LIN {X 0,Y 683.026,Z 572.337,A -85,B 0,C 180,E1 -4274.214,E2 -4274.214} C_VEL
LIN {X 0,Y 683.001,Z 572.333,A -85,B 0,C 180,E1 -4276.73,E2 -4276.73} C_VEL
LIN {X 0,Y 683.022,Z 572.332,A -85,B 0,C 180,E1 -4279.365,E2 -4279.365} C_VEL
LIN {X 0,Y 682.974,Z 572.347,A -85,B 0,C 180,E1 -4282.023,E2 -4282.023} C_VEL
LIN {X 0,Y 683,Z 572.34,A -85,B 0,C 180,E1 -4284.229,E2 -4284.229} C_VEL
LIN {X 0,Y 682.988,Z 572.339,A -85,B 0,C 180,E1 -4286.372,E2 -4286.372} C_VEL
LIN {X 0,Y 683.015,Z 572.334,A -85,B 0,C 180,E1 -4288.466,E2 -4288.466} C_VEL
LIN {X 0,Y 682.998,Z 572.334,A -85,B 0,C 180,E1 -4291.184,E2 -4291.184} C_VEL
LIN {X 0,Y 682.965,Z 572.347,A -85,B 0,C 180,E1 -4293.832,E2 -4293.832} C_VEL
LIN {X 0,Y 682.994,Z 572.345,A -85,B 0,C 180,E1 -4295.887,E2 -4295.887} C_VEL
LIN {X 0,Y 683.01,Z 572.336,A -85,B 0,C 180,E1 -4298.335,E2 -4298.335} C_VEL
LIN {X 0,Y 683.033,Z 572.329,A -85,B 0,C 180,E1 -4300.843,E2 -4300.843} C_VEL
LIN {X 0,Y 682.992,Z 572.336,A -85,B 0,C 180,E1 -4303.313,E2 -4303.313} C_VEL
LIN {X 0,Y 682.988,Z 572.343,A -85,B 0,C 180,E1 -4305.751,E2 -4305.751} C_VEL
LIN {X 0,Y 683.006,Z 572.34,A -85,B 0,C 180,E1 -4308.165,E2 -4308.165} C_VEL
LIN {X 0,Y 683.046,Z 572.329,A -85,B 0,C 180,E1 -4310.557,E2 -4310.557} C_VEL
LIN {X 0,Y 683.043,Z 572.328,A -85,B 0,C 180,E1 -4312.932,E2 -4312.932} C_VEL
LIN {X 0,Y 683.01,Z 572.332,A -85,B 0,C 180,E1 -4314.704,E2 -4314.704} C_VEL
LIN {X 0,Y 682.952,Z 572.342,A -85,B 0,C 180,E1 -4316.472,E2 -4316.472} C_VEL
LIN {X 0,Y 683.121,Z 572.318,A -85,B 0,C 180,E1 -4318.825,E2 -4318.825} C_VEL
LIN {X 0,Y 683.102,Z 572.329,A -85,B 0,C 180,E1 -4321.763,E2 -4321.763} C_VEL
LIN {X 0,Y 683.07,Z 572.325,A -85,B 0,C 180,E1 -4324.706,E2 -4324.706} C_VEL
LIN {X 0,Y 683.037,Z 572.328,A -85,B 0,C 180,E1 -4327.069,E2 -4327.069} C_VEL
LIN {X 0,Y 683.062,Z 572.336,A -85,B 0,C 180,E1 -4330.04,E2 -4330.04} C_VEL
LIN {X 0,Y 683.032,Z 572.329,A -85,B 0,C 180,E1 -4333.039,E2 -4333.039} C_VEL
LIN {X 0,Y 683.005,Z 572.336,A -85,B 0,C 180,E1 -4335.464,E2 -4335.464} C_VEL
LIN {X 0,Y 682.987,Z 572.347,A -85,B 0,C 180,E1 -4337.919,E2 -4337.919} C_VEL
LIN {X 0,Y 682.965,Z 572.346,A -85,B 0,C 180,E1 -4339.782,E2 -4339.782} C_VEL
LIN {X 0,Y 682.975,Z 572.337,A -85,B 0,C 180,E1 -4342.628,E2 -4342.628} C_VEL
LIN {X 0,Y 682.991,Z 572.334,A -85,B 0,C 180,E1 -4344.865,E2 -4344.865} C_VEL
LIN {X 0,Y 682.98,Z 572.339,A -85,B 0,C 180,E1 -4347.484,E2 -4347.484} C_VEL
LIN {X 0,Y 682.979,Z 572.34,A -85,B 0,C 180,E1 -4349.49,E2 -4349.49} C_VEL
LIN {X 0,Y 682.971,Z 572.343,A -85,B 0,C 180,E1 -4352.229,E2 -4352.229} C_VEL
LIN {X 0,Y 682.965,Z 572.342,A -85,B 0,C 180,E1 -4354.338,E2 -4354.338} C_VEL
LIN {X 0,Y 682.944,Z 572.34,A -85,B 0,C 180,E1 -4356.871,E2 -4356.871} C_VEL
LIN {X 0,Y 682.965,Z 572.338,A -85,B 0,C 180,E1 -4358.79,E2 -4358.79} C_VEL
LIN {X 0,Y 682.959,Z 572.343,A -85,B 0,C 180,E1 -4361.523,E2 -4361.523} C_VEL
LIN {X 0,Y 682.988,Z 572.341,A -85,B 0,C 180,E1 -4364.217,E2 -4364.217} C_VEL
LIN {X 0,Y 682.936,Z 572.341,A -85,B 0,C 180,E1 -4366.736,E2 -4366.736} C_VEL
LIN {X 0,Y 682.97,Z 572.339,A -85,B 0,C 180,E1 -4369.37,E2 -4369.37} C_VEL
LIN {X 0,Y 682.965,Z 572.345,A -85,B 0,C 180,E1 -4372.158,E2 -4372.158} C_VEL
LIN {X 0,Y 682.961,Z 572.338,A -85,B 0,C 180,E1 -4374.947,E2 -4374.947} C_VEL
LIN {X 0,Y 682.985,Z 572.336,A -85,B 0,C 180,E1 -4377.242,E2 -4377.242} C_VEL
LIN {X 0,Y 682.949,Z 572.349,A -85,B 0,C 180,E1 -4379.831,E2 -4379.831} C_VEL
LIN {X 0,Y 682.954,Z 572.341,A -85,B 0,C 180,E1 -4382.515,E2 -4382.515} C_VEL
LIN {X 0,Y 682.986,Z 572.337,A -85,B 0,C 180,E1 -4385.135,E2 -4385.135} C_VEL
LIN {X 0,Y 682.994,Z 572.346,A -85,B 0,C 180,E1 -4388.215,E2 -4388.215} C_VEL
LIN {X 0,Y 683.856,Z 577.659,A -85,B 0,C 180,E1 -4388.993,E2 -4388.993} C_VEL
LIN {X 0,Y 683.698,Z 593.941,A -85,B 0,C 180,E1 -4391.173,E2 -4391.173} C_VEL
LIN {X 0,Y 683.385,Z 612.574,A -85,B 0,C 180,E1 -4393.629,E2 -4393.629} C_VEL
LIN {X 0,Y 683.159,Z 631.189,A -85,B 0,C 180,E1 -4396.058,E2 -4396.058} C_VEL
LIN {X 0,Y 682.934,Z 649.485,A -85,B 0,C 180,E1 -4398.426,E2 -4398.426} C_VEL
LIN {X 0,Y 683.89,Z 658.24,A -85,B 0,C 180,E1 -4398.536,E2 -4398.536} C_VEL
LIN {X 0,Y 683.613,Z 755.729,A -85,B 0,C 180,E1 -4399.57,E2 -4399.57} C_VEL
LIN {X 0,Y 683.524,Z 765.358,A -85,B 0,C 180,E1 -4399.735,E2 -4399.735} C_VEL
LIN {X 0,Y 683.504,Z 776.178,A -85,B 0,C 180,E1 -4400.004,E2 -4400.004} C_VEL
LIN {X 0,Y 683.404,Z 786.265,A -85,B 0,C 180,E1 -4400.338,E2 -4400.338} C_VEL
LIN {X 0,Y 683.279,Z 796.757,A -85,B 0,C 180,E1 -4400.783,E2 -4400.783} C_VEL
LIN {X 0,Y 683.151,Z 806.601,A -85,B 0,C 180,E1 -4401.302,E2 -4401.302} C_VEL
LIN {X 0,Y 682.995,Z 814.812,A -85,B 0,C 180,E1 -4401.819,E2 -4401.819} C_VEL
LIN {X 0,Y 682.831,Z 823.576,A -85,B 0,C 180,E1 -4402.485,E2 -4402.485} C_VEL
LIN {X 0,Y 682.732,Z 831.633,A -85,B 0,C 180,E1 -4403.224,E2 -4403.224} C_VEL
LIN {X 0,Y 682.647,Z 838.345,A -85,B 0,C 180,E1 -4403.963,E2 -4403.963} C_VEL
LIN {X 0,Y 682.561,Z 843.958,A -85,B 0,C 180,E1 -4404.701,E2 -4404.701} C_VEL
LIN {X 0,Y 682.519,Z 849.404,A -85,B 0,C 180,E1 -4405.586,E2 -4405.586} C_VEL
LIN {X 0,Y 682.471,Z 853.686,A -85,B 0,C 180,E1 -4406.47,E2 -4406.47} C_VEL
LIN {X 0,Y 682.508,Z 855.979,A -85,B 0,C 180,E1 -4407.059,E2 -4407.059} C_VEL
LIN {X 0,Y 682.422,Z 859.189,A -85,B 0,C 180,E1 -4408.236,E2 -4408.236} C_VEL
LIN {X 0,Y 682.405,Z 860.148,A -85,B 0,C 180,E1 -4408.824,E2 -4408.824} C_VEL
LIN {X 0,Y 682.375,Z 861,A -85,B 0,C 180,E1 -4410,E2 -4410} C_VEL
LIN {X 0,Y 682.406,Z 860.149,A -85,B 0,C 180,E1 -4411.176,E2 -4411.176} C_VEL
LIN {X 0,Y 682.423,Z 859.191,A -85,B 0,C 180,E1 -4411.765,E2 -4411.765} C_VEL
LIN {X 0,Y 682.508,Z 855.981,A -85,B 0,C 180,E1 -4412.941,E2 -4412.941} C_VEL
LIN {X 0,Y 682.475,Z 852.425,A -85,B 0,C 180,E1 -4413.825,E2 -4413.825} C_VEL
LIN {X 0,Y 682.558,Z 847.764,A -85,B 0,C 180,E1 -4414.709,E2 -4414.709} C_VEL
LIN {X 0,Y 682.601,Z 841.063,A -85,B 0,C 180,E1 -4415.694,E2 -4415.694} C_VEL
LIN {X 0,Y 682.667,Z 834.458,A -85,B 0,C 180,E1 -4416.481,E2 -4416.481} C_VEL
LIN {X 0,Y 682.799,Z 826.966,A -85,B 0,C 180,E1 -4417.219,E2 -4417.219} C_VEL
LIN {X 0,Y 682.918,Z 818.879,A -85,B 0,C 180,E1 -4417.885,E2 -4417.885} C_VEL
LIN {X 0,Y 683.048,Z 810.276,A -85,B 0,C 180,E1 -4418.477,E2 -4418.477} C_VEL
LIN {X 0,Y 683.207,Z 801.24,A -85,B 0,C 180,E1 -4418.995,E2 -4418.995} C_VEL
LIN {X 0,Y 683.361,Z 791.852,A -85,B 0,C 180,E1 -4419.439,E2 -4419.439} C_VEL
LIN {X 0,Y 683.439,Z 780.985,A -85,B 0,C 180,E1 -4419.848,E2 -4419.848} C_VEL
LIN {X 0,Y 683.513,Z 770.389,A -85,B 0,C 180,E1 -4420.152,E2 -4420.152} C_VEL
LIN {X 0,Y 683.657,Z 759.149,A -85,B 0,C 180,E1 -4420.38,E2 -4420.38} C_VEL
LIN {X 0,Y 683.695,Z 742.553,A -85,B 0,C 180,E1 -4420.584,E2 -4420.584} C_VEL
LIN {X 0,Y 683.821,Z 656.435,A -85,B 0,C 180,E1 -4421.484,E2 -4421.484} C_VEL
LIN {X 0,Y 682.934,Z 649.483,A -85,B 0,C 180,E1 -4421.575,E2 -4421.575} C_VEL
LIN {X 0,Y 683.16,Z 631.148,A -85,B 0,C 180,E1 -4423.943,E2 -4423.943} C_VEL
LIN {X 0,Y 683.411,Z 611.307,A -85,B 0,C 180,E1 -4426.524,E2 -4426.524} C_VEL
LIN {X 0,Y 683.768,Z 589.908,A -85,B 0,C 180,E1 -4429.339,E2 -4429.339} C_VEL
LIN {X 0,Y 683.834,Z 577.443,A -85,B 0,C 180,E1 -4431.008,E2 -4431.008} C_VEL
LIN {X 0,Y 682.983,Z 572.347,A -85,B 0,C 180,E1 -4431.746,E2 -4431.746} C_VEL
LIN {X 0,Y 682.954,Z 572.348,A -85,B 0,C 180,E1 -4434.22,E2 -4434.22} C_VEL
LIN {X 0,Y 682.968,Z 572.341,A -85,B 0,C 180,E1 -4436.841,E2 -4436.841} C_VEL
LIN {X 0,Y 682.969,Z 572.347,A -85,B 0,C 180,E1 -4439.491,E2 -4439.491} C_VEL
LIN {X 0,Y 682.972,Z 572.341,A -85,B 0,C 180,E1 -4442.229,E2 -4442.229} C_VEL
LIN {X 0,Y 682.979,Z 572.338,A -85,B 0,C 180,E1 -4444.87,E2 -4444.87} C_VEL
LIN {X 0,Y 682.963,Z 572.344,A -85,B 0,C 180,E1 -4447.236,E2 -4447.236} C_VEL
LIN {X 0,Y 682.955,Z 572.345,A -85,B 0,C 180,E1 -4449.717,E2 -4449.717} C_VEL
LIN {X 0,Y 682.985,Z 572.339,A -85,B 0,C 180,E1 -4451.807,E2 -4451.807} C_VEL
LIN {X 0,Y 682.996,Z 572.335,A -85,B 0,C 180,E1 -4454.217,E2 -4454.217} C_VEL
LIN {X 0,Y 683.006,Z 572.337,A -85,B 0,C 180,E1 -4456.73,E2 -4456.73} C_VEL
LIN {X 0,Y 683.028,Z 572.339,A -85,B 0,C 180,E1 -4459.365,E2 -4459.365} C_VEL
LIN {X 0,Y 682.977,Z 572.338,A -85,B 0,C 180,E1 -4462.157,E2 -4462.157} C_VEL
LIN {X 0,Y 683.018,Z 572.342,A -85,B 0,C 180,E1 -4464.95,E2 -4464.95} C_VEL
LIN {X 0,Y 683.017,Z 572.332,A -85,B 0,C 180,E1 -4467.773,E2 -4467.773} C_VEL
LIN {X 0,Y 682.996,Z 572.334,A -85,B 0,C 180,E1 -4469.833,E2 -4469.833} C_VEL
LIN {X 0,Y 683.027,Z 572.331,A -85,B 0,C 180,E1 -4471.876,E2 -4471.876} C_VEL
LIN {X 0,Y 682.998,Z 572.343,A -85,B 0,C 180,E1 -4474.486,E2 -4474.486} C_VEL
LIN {X 0,Y 683,Z 572.339,A -85,B 0,C 180,E1 -4477.064,E2 -4477.064} C_VEL
LIN {X 0,Y 682.981,Z 572.339,A -85,B 0,C 180,E1 -4479.592,E2 -4479.592} C_VEL
LIN {X 0,Y 683.01,Z 572.335,A -85,B 0,C 180,E1 -4481.463,E2 -4481.463} C_VEL
LIN {X 0,Y 682.992,Z 572.34,A -85,B 0,C 180,E1 -4483.925,E2 -4483.925} C_VEL
LIN {X 0,Y 683.015,Z 572.344,A -85,B 0,C 180,E1 -4486.357,E2 -4486.357} C_VEL
LIN {X 0,Y 683.015,Z 572.338,A -85,B 0,C 180,E1 -4488.764,E2 -4488.764} C_VEL
LIN {X 0,Y 683.058,Z 572.423,A -85,B 0,C 180,E1 -4490.929,E2 -4490.929} C_VEL
LIN {X 0,Y 683.487,Z 579.381,A -85,B 0,C 180,E1 -4492.048,E2 -4492.048} C_VEL
LIN {X 0,Y 683.242,Z 596.262,A -85,B 0,C 180,E1 -4494.706,E2 -4494.706} C_VEL
LIN {X 0,Y 682.99,Z 609.521,A -85,B 0,C 180,E1 -4496.766,E2 -4496.766} C_VEL
LIN {X 0,Y 682.853,Z 620.602,A -85,B 0,C 180,E1 -4498.475,E2 -4498.475} C_VEL
LIN {X 0,Y 683.914,Z 628.858,A -85,B 0,C 180,E1 -4498.588,E2 -4498.588} C_VEL
LIN {X 0,Y 683.517,Z 727.56,A -85,B 0,C 180,E1 -4499.633,E2 -4499.633} C_VEL
LIN {X 0,Y 683.418,Z 740.394,A -85,B 0,C 180,E1 -4499.89,E2 -4499.89} C_VEL
LIN {X 0,Y 683.336,Z 752.881,A -85,B 0,C 180,E1 -4500.257,E2 -4500.257} C_VEL
LIN {X 0,Y 683.323,Z 764.89,A -85,B 0,C 180,E1 -4500.734,E2 -4500.734} C_VEL
LIN {X 0,Y 683.123,Z 776.26,A -85,B 0,C 180,E1 -4501.322,E2 -4501.322} C_VEL
LIN {X 0,Y 682.987,Z 786.525,A -85,B 0,C 180,E1 -4501.983,E2 -4501.983} C_VEL
LIN {X 0,Y 682.762,Z 795.042,A -85,B 0,C 180,E1 -4502.646,E2 -4502.646} C_VEL
LIN {X 0,Y 682.683,Z 802.781,A -85,B 0,C 180,E1 -4503.382,E2 -4503.382} C_VEL
LIN {X 0,Y 682.531,Z 810.48,A -85,B 0,C 180,E1 -4504.267,E2 -4504.267} C_VEL
LIN {X 0,Y 682.532,Z 815.691,A -85,B 0,C 180,E1 -4505.004,E2 -4505.004} C_VEL
LIN {X 0,Y 682.498,Z 820.823,A -85,B 0,C 180,E1 -4505.89,E2 -4505.89} C_VEL
LIN {X 0,Y 682.465,Z 824.783,A -85,B 0,C 180,E1 -4506.778,E2 -4506.778} C_VEL
LIN {X 0,Y 682.403,Z 827.744,A -85,B 0,C 180,E1 -4507.668,E2 -4507.668} C_VEL
LIN {X 0,Y 682.391,Z 829.173,A -85,B 0,C 180,E1 -4508.262,E2 -4508.262} C_VEL
LIN {X 0,Y 682.414,Z 830.191,A -85,B 0,C 180,E1 -4508.856,E2 -4508.856} C_VEL
LIN {X 0,Y 682.438,Z 831,A -85,B 0,C 180,E1 -4510.048,E2 -4510.048} C_VEL
LIN {X 0,Y 682.389,Z 830.173,A -85,B 0,C 180,E1 -4511.246,E2 -4511.246} C_VEL
LIN {X 0,Y 682.396,Z 829.138,A -85,B 0,C 180,E1 -4511.846,E2 -4511.846} C_VEL
LIN {X 0,Y 682.448,Z 826.515,A -85,B 0,C 180,E1 -4512.824,E2 -4512.824} C_VEL
LIN {X 0,Y 682.443,Z 823.402,A -85,B 0,C 180,E1 -4513.654,E2 -4513.654} C_VEL
LIN {X 0,Y 682.509,Z 818.861,A -85,B 0,C 180,E1 -4514.562,E2 -4514.562} C_VEL
LIN {X 0,Y 682.562,Z 813.1,A -85,B 0,C 180,E1 -4515.474,E2 -4515.474} C_VEL
LIN {X 0,Y 682.66,Z 805.78,A -85,B 0,C 180,E1 -4516.389,E2 -4516.389} C_VEL
LIN {X 0,Y 682.765,Z 798.238,A -85,B 0,C 180,E1 -4517.154,E2 -4517.154} C_VEL
LIN {X 0,Y 682.922,Z 789.106,A -85,B 0,C 180,E1 -4517.92,E2 -4517.92} C_VEL
LIN {X 0,Y 683.022,Z 778.927,A -85,B 0,C 180,E1 -4518.614,E2 -4518.614} C_VEL
LIN {X 0,Y 683.166,Z 769.09,A -85,B 0,C 180,E1 -4519.153,E2 -4519.153} C_VEL
LIN {X 0,Y 683.38,Z 757.902,A -85,B 0,C 180,E1 -4519.651,E2 -4519.651} C_VEL
LIN {X 0,Y 683.455,Z 746.324,A -85,B 0,C 180,E1 -4520.04,E2 -4520.04} C_VEL
LIN {X 0,Y 683.581,Z 733.577,A -85,B 0,C 180,E1 -4520.349,E2 -4520.349} C_VEL
LIN {X 0,Y 683.672,Z 720.861,A -85,B 0,C 180,E1 -4520.542,E2 -4520.542} C_VEL
LIN {X 0,Y 683.853,Z 627.908,A -85,B 0,C 180,E1 -4521.513,E2 -4521.513} C_VEL
LIN {X 0,Y 682.833,Z 620.616,A -85,B 0,C 180,E1 -4521.611,E2 -4521.611} C_VEL
LIN {X 0,Y 682.975,Z 608.393,A -85,B 0,C 180,E1 -4523.492,E2 -4523.492} C_VEL
LIN {X 0,Y 682.356,Z 605.665,A -85,B 0,C 180,E1 -4523.928,E2 -4523.928} C_VEL
LIN {X 0,Y 676.758,Z 597.294,A -85,B 0,C 180,E1 -4525.373,E2 -4525.373} C_VEL
LIN {X 0,Y 676.16,Z 594.582,A -85,B 0,C 180,E1 -4525.816,E2 -4525.816} C_VEL
LIN {X 0,Y 676.414,Z 577.967,A -85,B 0,C 180,E1 -4528.446,E2 -4528.446} C_VEL
LIN {X 0,Y 675.969,Z 573.219,A -85,B 0,C 180,E1 -4529.233,E2 -4529.233} C_VEL
LIN {X 0,Y 675.971,Z 573.212,A -85,B 0,C 180,E1 -4531.205,E2 -4531.205} C_VEL
LIN {X 0,Y 675.962,Z 573.221,A -85,B 0,C 180,E1 -4534.025,E2 -4534.025} C_VEL
LIN {X 0,Y 675.942,Z 573.219,A -85,B 0,C 180,E1 -4536.204,E2 -4536.204} C_VEL
LIN {X 0,Y 675.938,Z 573.213,A -85,B 0,C 180,E1 -4538.996,E2 -4538.996} C_VEL
LIN {X 0,Y 675.972,Z 573.216,A -85,B 0,C 180,E1 -4541.749,E2 -4541.749} C_VEL
LIN {X 0,Y 675.985,Z 573.211,A -85,B 0,C 180,E1 -4544.359,E2 -4544.359} C_VEL
LIN {X 0,Y 675.946,Z 573.212,A -85,B 0,C 180,E1 -4546.849,E2 -4546.849} C_VEL
LIN {X 0,Y 675.967,Z 573.21,A -85,B 0,C 180,E1 -4549.246,E2 -4549.246} C_VEL
LIN {X 0,Y 675.937,Z 573.225,A -85,B 0,C 180,E1 -4551.957,E2 -4551.957} C_VEL
LIN {X 0,Y 675.946,Z 573.214,A -85,B 0,C 180,E1 -4554.528,E2 -4554.528} C_VEL
LIN {X 0,Y 675.946,Z 573.212,A -85,B 0,C 180,E1 -4557.071,E2 -4557.071} C_VEL
LIN {X 0,Y 676.001,Z 573.209,A -85,B 0,C 180,E1 -4559.488,E2 -4559.488} C_VEL
LIN {X 0,Y 675.948,Z 573.219,A -85,B 0,C 180,E1 -4562.205,E2 -4562.205} C_VEL
LIN {X 0,Y 675.945,Z 573.212,A -85,B 0,C 180,E1 -4564.858,E2 -4564.858} C_VEL
LIN {X 0,Y 675.976,Z 573.211,A -85,B 0,C 180,E1 -4567.456,E2 -4567.456} C_VEL
LIN {X 0,Y 675.936,Z 573.224,A -85,B 0,C 180,E1 -4570.003,E2 -4570.003} C_VEL
LIN {X 0,Y 675.997,Z 573.208,A -85,B 0,C 180,E1 -4572.513,E2 -4572.513} C_VEL
LIN {X 0,Y 675.997,Z 573.205,A -85,B 0,C 180,E1 -4574.987,E2 -4574.987} C_VEL
LIN {X 0,Y 675.997,Z 573.208,A -85,B 0,C 180,E1 -4577.432,E2 -4577.432} C_VEL
LIN {X 0,Y 676.01,Z 573.207,A -85,B 0,C 180,E1 -4580.457,E2 -4580.457} C_VEL
LIN {X 0,Y 676.011,Z 573.204,A -85,B 0,C 180,E1 -4582.857,E2 -4582.857} C_VEL
LIN {X 0,Y 676.046,Z 573.2,A -85,B 0,C 180,E1 -4585.245,E2 -4585.245} C_VEL
LIN {X 0,Y 676.106,Z 573.192,A -85,B 0,C 180,E1 -4588.813,E2 -4588.813} C_VEL
LIN {X 0,Y 676.086,Z 573.203,A -85,B 0,C 180,E1 -4591.781,E2 -4591.781} C_VEL
LIN {X 0,Y 676.046,Z 573.2,A -85,B 0,C 180,E1 -4594.754,E2 -4594.754} C_VEL
LIN {X 0,Y 676.011,Z 573.204,A -85,B 0,C 180,E1 -4597.142,E2 -4597.142} C_VEL
LIN {X 0,Y 675.986,Z 573.215,A -85,B 0,C 180,E1 -4600.146,E2 -4600.146} C_VEL
LIN {X 0,Y 676.012,Z 573.204,A -85,B 0,C 180,E1 -4603.176,E2 -4603.176} C_VEL
LIN {X 0,Y 676.008,Z 573.21,A -85,B 0,C 180,E1 -4605.628,E2 -4605.628} C_VEL
LIN {X 0,Y 675.976,Z 573.217,A -85,B 0,C 180,E1 -4608.111,E2 -4608.111} C_VEL
LIN {X 0,Y 675.954,Z 573.212,A -85,B 0,C 180,E1 -4610.629,E2 -4610.629} C_VEL
LIN {X 0,Y 675.962,Z 573.21,A -85,B 0,C 180,E1 -4613.189,E2 -4613.189} C_VEL
LIN {X 0,Y 675.928,Z 573.223,A -85,B 0,C 180,E1 -4615.8,E2 -4615.8} C_VEL
LIN {X 0,Y 675.958,Z 573.216,A -85,B 0,C 180,E1 -4618.263,E2 -4618.263} C_VEL
LIN {X 0,Y 675.995,Z 573.206,A -85,B 0,C 180,E1 -4620.682,E2 -4620.682} C_VEL
LIN {X 0,Y 675.96,Z 573.212,A -85,B 0,C 180,E1 -4623.312,E2 -4623.312} C_VEL
LIN {X 0,Y 675.978,Z 573.217,A -85,B 0,C 180,E1 -4626.077,E2 -4626.077} C_VEL
LIN {X 0,Y 675.937,Z 573.213,A -85,B 0,C 180,E1 -4628.997,E2 -4628.997} C_VEL
LIN {X 0,Y 675.97,Z 573.217,A -85,B 0,C 180,E1 -4631.75,E2 -4631.75} C_VEL
LIN {X 0,Y 675.984,Z 573.211,A -85,B 0,C 180,E1 -4634.36,E2 -4634.36} C_VEL
LIN {X 0,Y 675.944,Z 573.212,A -85,B 0,C 180,E1 -4636.85,E2 -4636.85} C_VEL
LIN {X 0,Y 675.966,Z 573.21,A -85,B 0,C 180,E1 -4639.246,E2 -4639.246} C_VEL
LIN {X 0,Y 675.938,Z 573.225,A -85,B 0,C 180,E1 -4641.957,E2 -4641.957} C_VEL
LIN {X 0,Y 675.946,Z 573.214,A -85,B 0,C 180,E1 -4644.529,E2 -4644.529} C_VEL
LIN {X 0,Y 675.946,Z 573.212,A -85,B 0,C 180,E1 -4647.072,E2 -4647.072} C_VEL
LIN {X 0,Y 676.002,Z 573.209,A -85,B 0,C 180,E1 -4649.489,E2 -4649.489} C_VEL
LIN {X 0,Y 675.944,Z 573.219,A -85,B 0,C 180,E1 -4652.205,E2 -4652.205} C_VEL
LIN {X 0,Y 675.947,Z 573.212,A -85,B 0,C 180,E1 -4654.859,E2 -4654.859} C_VEL
LIN {X 0,Y 675.977,Z 573.211,A -85,B 0,C 180,E1 -4657.456,E2 -4657.456} C_VEL
LIN {X 0,Y 675.937,Z 573.224,A -85,B 0,C 180,E1 -4660.004,E2 -4660.004} C_VEL
LIN {X 0,Y 675.958,Z 573.213,A -85,B 0,C 180,E1 -4662.512,E2 -4662.512} C_VEL
LIN {X 0,Y 675.945,Z 573.212,A -85,B 0,C 180,E1 -4664.986,E2 -4664.986} C_VEL
LIN {X 0,Y 675.984,Z 573.21,A -85,B 0,C 180,E1 -4667.432,E2 -4667.432} C_VEL
LIN {X 0,Y 676.031,Z 573.212,A -85,B 0,C 180,E1 -4669.855,E2 -4669.855} C_VEL
LIN {X 0,Y 676.011,Z 573.204,A -85,B 0,C 180,E1 -4672.858,E2 -4672.858} C_VEL
LIN {X 0,Y 676.013,Z 573.205,A -85,B 0,C 180,E1 -4675.245,E2 -4675.245} C_VEL
LIN {X 0,Y 676.107,Z 573.198,A -85,B 0,C 180,E1 -4678.219,E2 -4678.219} C_VEL
LIN {X 0,Y 676.095,Z 573.194,A -85,B 0,C 180,E1 -4681.187,E2 -4681.187} C_VEL
LIN {X 0,Y 676.053,Z 573.206,A -85,B 0,C 180,E1 -4684.159,E2 -4684.159} C_VEL
LIN {X 0,Y 676.026,Z 573.204,A -85,B 0,C 180,E1 -4686.545,E2 -4686.545} C_VEL
LIN {X 0,Y 676.015,Z 573.208,A -85,B 0,C 180,E1 -4689.543,E2 -4689.543} C_VEL
LIN {X 0,Y 675.944,Z 573.224,A -85,B 0,C 180,E1 -4691.961,E2 -4691.961} C_VEL
LIN {X 0,Y 675.945,Z 573.216,A -85,B 0,C 180,E1 -4694.401,E2 -4694.401} C_VEL
LIN {X 0,Y 675.928,Z 573.214,A -85,B 0,C 180,E1 -4696.867,E2 -4696.867} C_VEL
LIN {X 0,Y 675.937,Z 573.216,A -85,B 0,C 180,E1 -4699.44,E2 -4699.44} C_VEL
LIN {X 0,Y 675.945,Z 573.223,A -85,B 0,C 180,E1 -4701.904,E2 -4701.904} C_VEL
LIN {X 0,Y 675.937,Z 573.215,A -85,B 0,C 180,E1 -4704.488,E2 -4704.488} C_VEL
LIN {X 0,Y 675.959,Z 573.211,A -85,B 0,C 180,E1 -4707.125,E2 -4707.125} C_VEL
LIN {X 0,Y 675.954,Z 573.215,A -85,B 0,C 180,E1 -4709.491,E2 -4709.491} C_VEL
LIN {X 0,Y 675.917,Z 573.227,A -85,B 0,C 180,E1 -4711.905,E2 -4711.905} C_VEL
LIN {X 0,Y 675.934,Z 573.224,A -85,B 0,C 180,E1 -4714.027,E2 -4714.027} C_VEL
LIN {X 0,Y 675.917,Z 573.222,A -85,B 0,C 180,E1 -4716.206,E2 -4716.206} C_VEL
LIN {X 0,Y 675.928,Z 573.217,A -85,B 0,C 180,E1 -4718.445,E2 -4718.445} C_VEL
LIN {X 0,Y 675.908,Z 573.217,A -85,B 0,C 180,E1 -4720.843,E2 -4720.843} C_VEL
LIN {X 0,Y 675.915,Z 573.22,A -85,B 0,C 180,E1 -4723.498,E2 -4723.498} C_VEL
LIN {X 0,Y 675.938,Z 573.223,A -85,B 0,C 180,E1 -4726.029,E2 -4726.029} C_VEL
LIN {X 0,Y 675.912,Z 573.219,A -85,B 0,C 180,E1 -4728.453,E2 -4728.453} C_VEL
LIN {X 0,Y 675.922,Z 573.215,A -85,B 0,C 180,E1 -4731.006,E2 -4731.006} C_VEL
LIN {X 0,Y 675.912,Z 573.225,A -85,B 0,C 180,E1 -4733.794,E2 -4733.794} C_VEL
LIN {X 0,Y 675.934,Z 573.225,A -85,B 0,C 180,E1 -4735.997,E2 -4735.997} C_VEL
LIN {X 0,Y 675.917,Z 573.223,A -85,B 0,C 180,E1 -4738.185,E2 -4738.185} C_VEL
LIN {X 0,Y 675.911,Z 573.216,A -85,B 0,C 180,E1 -4740.853,E2 -4740.853} C_VEL
LIN {X 0,Y 675.895,Z 573.223,A -85,B 0,C 180,E1 -4743.537,E2 -4743.537} C_VEL
LIN {X 0,Y 675.916,Z 573.227,A -85,B 0,C 180,E1 -4745.774,E2 -4745.774} C_VEL
LIN {X 0,Y 675.945,Z 573.231,A -85,B 0,C 180,E1 -4748.136,E2 -4748.136} C_VEL
LIN {X 0,Y 676.938,Z 579.896,A -85,B 0,C 180,E1 -4749.085,E2 -4749.085} C_VEL
LIN {X 0,Y 676.678,Z 598.495,A -85,B 0,C 180,E1 -4751.596,E2 -4751.596} C_VEL
LIN {X 0,Y 676.257,Z 619.451,A -85,B 0,C 180,E1 -4754.378,E2 -4754.378} C_VEL
LIN {X 0,Y 676.033,Z 638.061,A -85,B 0,C 180,E1 -4756.824,E2 -4756.824} C_VEL
LIN {X 0,Y 675.918,Z 649.673,A -85,B 0,C 180,E1 -4758.313,E2 -4758.313} C_VEL
LIN {X 0,Y 676.947,Z 659.587,A -85,B 0,C 180,E1 -4758.435,E2 -4758.435} C_VEL
LIN {X 0,Y 676.655,Z 754.661,A -85,B 0,C 180,E1 -4759.451,E2 -4759.451} C_VEL
LIN {X 0,Y 676.534,Z 764.965,A -85,B 0,C 180,E1 -4759.623,E2 -4759.623} C_VEL
LIN {X 0,Y 676.501,Z 776.042,A -85,B 0,C 180,E1 -4759.9,E2 -4759.9} C_VEL
LIN {X 0,Y 676.405,Z 786.18,A -85,B 0,C 180,E1 -4760.237,E2 -4760.237} C_VEL
LIN {X 0,Y 676.284,Z 796.718,A -85,B 0,C 180,E1 -4760.687,E2 -4760.687} C_VEL
LIN {X 0,Y 676.116,Z 806.595,A -85,B 0,C 180,E1 -4761.21,E2 -4761.21} C_VEL
LIN {X 0,Y 675.972,Z 814.81,A -85,B 0,C 180,E1 -4761.734,E2 -4761.734} C_VEL
LIN {X 0,Y 675.786,Z 823.574,A -85,B 0,C 180,E1 -4762.406,E2 -4762.406} C_VEL
LIN {X 0,Y 675.674,Z 831.632,A -85,B 0,C 180,E1 -4763.153,E2 -4763.153} C_VEL
LIN {X 0,Y 675.583,Z 838.344,A -85,B 0,C 180,E1 -4763.9,E2 -4763.9} C_VEL
LIN {X 0,Y 675.481,Z 843.958,A -85,B 0,C 180,E1 -4764.645,E2 -4764.645} C_VEL
LIN {X 0,Y 675.452,Z 849.404,A -85,B 0,C 180,E1 -4765.539,E2 -4765.539} C_VEL
LIN {X 0,Y 675.373,Z 853.686,A -85,B 0,C 180,E1 -4766.432,E2 -4766.432} C_VEL
LIN {X 0,Y 675.421,Z 855.98,A -85,B 0,C 180,E1 -4767.028,E2 -4767.028} C_VEL
LIN {X 0,Y 675.329,Z 859.188,A -85,B 0,C 180,E1 -4768.217,E2 -4768.217} C_VEL
LIN {X 0,Y 675.332,Z 860.146,A -85,B 0,C 180,E1 -4768.812,E2 -4768.812} C_VEL
LIN {X 0,Y 675.295,Z 861,A -85,B 0,C 180,E1 -4770,E2 -4770} C_VEL
LIN {X 0,Y 675.332,Z 860.148,A -85,B 0,C 180,E1 -4771.189,E2 -4771.189} C_VEL
LIN {X 0,Y 675.329,Z 859.19,A -85,B 0,C 180,E1 -4771.783,E2 -4771.783} C_VEL
LIN {X 0,Y 675.421,Z 855.982,A -85,B 0,C 180,E1 -4772.972,E2 -4772.972} C_VEL
LIN {X 0,Y 675.385,Z 852.426,A -85,B 0,C 180,E1 -4773.865,E2 -4773.865} C_VEL
LIN {X 0,Y 675.479,Z 847.763,A -85,B 0,C 180,E1 -4774.759,E2 -4774.759} C_VEL
LIN {X 0,Y 675.516,Z 841.85,A -85,B 0,C 180,E1 -4775.653,E2 -4775.653} C_VEL
LIN {X 0,Y 675.602,Z 835.87,A -85,B 0,C 180,E1 -4776.399,E2 -4776.399} C_VEL
LIN {X 0,Y 675.744,Z 828.661,A -85,B 0,C 180,E1 -4777.145,E2 -4777.145} C_VEL
LIN {X 0,Y 675.859,Z 819.894,A -85,B 0,C 180,E1 -4777.893,E2 -4777.893} C_VEL
LIN {X 0,Y 676.032,Z 810.273,A -85,B 0,C 180,E1 -4778.566,E2 -4778.566} C_VEL
LIN {X 0,Y 676.179,Z 801.215,A -85,B 0,C 180,E1 -4779.089,E2 -4779.089} C_VEL
LIN {X 0,Y 676.361,Z 791.781,A -85,B 0,C 180,E1 -4779.538,E2 -4779.538} C_VEL
LIN {X 0,Y 676.448,Z 780.844,A -85,B 0,C 180,E1 -4779.95,E2 -4779.95} C_VEL
LIN {X 0,Y 676.504,Z 770.221,A -85,B 0,C 180,E1 -4780.257,E2 -4780.257} C_VEL
LIN {X 0,Y 676.671,Z 758.941,A -85,B 0,C 180,E1 -4780.486,E2 -4780.486} C_VEL
LIN {X 0,Y 676.71,Z 740.988,A -85,B 0,C 180,E1 -4780.706,E2 -4780.706} C_VEL
LIN {X 0,Y 676.87,Z 657.09,A -85,B 0,C 180,E1 -4781.59,E2 -4781.59} C_VEL
LIN {X 0,Y 675.882,Z 649.336,A -85,B 0,C 180,E1 -4781.697,E2 -4781.697} C_VEL
LIN {X 0,Y 676.101,Z 632.152,A -85,B 0,C 180,E1 -4783.938,E2 -4783.938} C_VEL
LIN {X 0,Y 676.35,Z 614.648,A -85,B 0,C 180,E1 -4786.238,E2 -4786.238} C_VEL
LIN {X 0,Y 676.678,Z 594.78,A -85,B 0,C 180,E1 -4788.873,E2 -4788.873} C_VEL
LIN {X 0,Y 676.843,Z 578.469,A -85,B 0,C 180,E1 -4791.077,E2 -4791.077} C_VEL
LIN {X 0,Y 675.951,Z 573.223,A -85,B 0,C 180,E1 -4791.824,E2 -4791.824} C_VEL
LIN {X 0,Y 675.908,Z 573.222,A -85,B 0,C 180,E1 -4794.489,E2 -4794.489} C_VEL
LIN {X 0,Y 675.907,Z 573.222,A -85,B 0,C 180,E1 -4797.128,E2 -4797.128} C_VEL
LIN {X 0,Y 675.903,Z 573.229,A -85,B 0,C 180,E1 -4799.83,E2 -4799.83} C_VEL
LIN {X 0,Y 675.917,Z 573.225,A -85,B 0,C 180,E1 -4801.905,E2 -4801.905} C_VEL
LIN {X 0,Y 675.937,Z 573.219,A -85,B 0,C 180,E1 -4804.027,E2 -4804.027} C_VEL
LIN {X 0,Y 675.938,Z 573.215,A -85,B 0,C 180,E1 -4806.204,E2 -4806.204} C_VEL
LIN {X 0,Y 675.931,Z 573.216,A -85,B 0,C 180,E1 -4808.995,E2 -4808.995} C_VEL
LIN {X 0,Y 675.969,Z 573.214,A -85,B 0,C 180,E1 -4811.749,E2 -4811.749} C_VEL
LIN {X 0,Y 675.943,Z 573.213,A -85,B 0,C 180,E1 -4814.356,E2 -4814.356} C_VEL
LIN {X 0,Y 675.952,Z 573.217,A -85,B 0,C 180,E1 -4816.85,E2 -4816.85} C_VEL
LIN {X 0,Y 675.972,Z 573.22,A -85,B 0,C 180,E1 -4819.246,E2 -4819.246} C_VEL
LIN {X 0,Y 675.942,Z 573.214,A -85,B 0,C 180,E1 -4821.957,E2 -4821.957} C_VEL
LIN {X 0,Y 675.969,Z 573.214,A -85,B 0,C 180,E1 -4824.53,E2 -4824.53} C_VEL
LIN {X 0,Y 675.955,Z 573.22,A -85,B 0,C 180,E1 -4827.071,E2 -4827.071} C_VEL
LIN {X 0,Y 676.007,Z 573.207,A -85,B 0,C 180,E1 -4829.488,E2 -4829.488} C_VEL
LIN {X 0,Y 675.949,Z 573.215,A -85,B 0,C 180,E1 -4832.205,E2 -4832.205} C_VEL
LIN {X 0,Y 675.952,Z 573.221,A -85,B 0,C 180,E1 -4834.858,E2 -4834.858} C_VEL
LIN {X 0,Y 675.982,Z 573.211,A -85,B 0,C 180,E1 -4837.456,E2 -4837.456} C_VEL
LIN {X 0,Y 675.941,Z 573.219,A -85,B 0,C 180,E1 -4840.003,E2 -4840.003} C_VEL
LIN {X 0,Y 675.963,Z 573.223,A -85,B 0,C 180,E1 -4842.512,E2 -4842.512} C_VEL
LIN {X 0,Y 675.948,Z 573.216,A -85,B 0,C 180,E1 -4844.986,E2 -4844.986} C_VEL
LIN {X 0,Y 675.988,Z 573.211,A -85,B 0,C 180,E1 -4847.432,E2 -4847.432} C_VEL
LIN {X 0,Y 676.034,Z 573.211,A -85,B 0,C 180,E1 -4849.855,E2 -4849.855} C_VEL
LIN {X 0,Y 676.005,Z 573.257,A -85,B 0,C 180,E1 -4850.833,E2 -4850.833} C_VEL
LIN {X 0,Y 676.493,Z 580.215,A -85,B 0,C 180,E1 -4851.965,E2 -4851.965} C_VEL
LIN {X 0,Y 676.231,Z 597.103,A -85,B 0,C 180,E1 -4854.651,E2 -4854.651} C_VEL
LIN {X 0,Y 675.963,Z 610.361,A -85,B 0,C 180,E1 -4856.733,E2 -4856.733} C_VEL
LIN {X 0,Y 675.79,Z 620.741,A -85,B 0,C 180,E1 -4858.348,E2 -4858.348} C_VEL
LIN {X 0,Y 676.987,Z 629.675,A -85,B 0,C 180,E1 -4858.481,E2 -4858.481} C_VEL
LIN {X 0,Y 676.524,Z 726.639,A -85,B 0,C 180,E1 -4859.518,E2 -4859.518} C_VEL
LIN {X 0,Y 676.434,Z 739.193,A -85,B 0,C 180,E1 -4859.759,E2 -4859.759} C_VEL
LIN {X 0,Y 676.339,Z 751.611,A -85,B 0,C 180,E1 -4860.111,E2 -4860.111} C_VEL
LIN {X 0,Y 676.307,Z 763.86,A -85,B 0,C 180,E1 -4860.593,E2 -4860.593} C_VEL
LIN {X 0,Y 676.132,Z 774.189,A -85,B 0,C 180,E1 -4861.113,E2 -4861.113} C_VEL
LIN {X 0,Y 675.957,Z 784.924,A -85,B 0,C 180,E1 -4861.781,E2 -4861.781} C_VEL
LIN {X 0,Y 675.717,Z 794.53,A -85,B 0,C 180,E1 -4862.525,E2 -4862.525} C_VEL
LIN {X 0,Y 675.628,Z 802.37,A -85,B 0,C 180,E1 -4863.269,E2 -4863.269} C_VEL
LIN {X 0,Y 675.459,Z 810.155,A -85,B 0,C 180,E1 -4864.163,E2 -4864.163} C_VEL
LIN {X 0,Y 675.443,Z 815.777,A -85,B 0,C 180,E1 -4864.964,E2 -4864.964} C_VEL
LIN {X 0,Y 675.421,Z 821.328,A -85,B 0,C 180,E1 -4865.952,E2 -4865.952} C_VEL
LIN {X 0,Y 675.367,Z 825.207,A -85,B 0,C 180,E1 -4866.85,E2 -4866.85} C_VEL
LIN {X 0,Y 675.298,Z 828.009,A -85,B 0,C 180,E1 -4867.749,E2 -4867.749} C_VEL
LIN {X 0,Y 675.316,Z 829.36,A -85,B 0,C 180,E1 -4868.349,E2 -4868.349} C_VEL
LIN {X 0,Y 675.315,Z 830.303,A -85,B 0,C 180,E1 -4868.95,E2 -4868.95} C_VEL
LIN {X 0,Y 675.351,Z 830.938,A -85,B 0,C 180,E1 -4869.836,E2 -4869.836} C_VEL
LIN {X 0,Y 675.321,Z 830.704,A -85,B 0,C 180,E1 -4870.76,E2 -4870.76} C_VEL
LIN {X 0,Y 675.286,Z 830.017,A -85,B 0,C 180,E1 -4871.366,E2 -4871.366} C_VEL
LIN {X 0,Y 675.318,Z 828.92,A -85,B 0,C 180,E1 -4871.972,E2 -4871.972} C_VEL
LIN {X 0,Y 675.361,Z 826.489,A -85,B 0,C 180,E1 -4872.86,E2 -4872.86} C_VEL
LIN {X 0,Y 675.354,Z 822.944,A -85,B 0,C 180,E1 -4873.8,E2 -4873.8} C_VEL
LIN {X 0,Y 675.445,Z 818.247,A -85,B 0,C 180,E1 -4874.718,E2 -4874.718} C_VEL
LIN {X 0,Y 675.504,Z 812.288,A -85,B 0,C 180,E1 -4875.64,E2 -4875.64} C_VEL
LIN {X 0,Y 675.6,Z 804.817,A -85,B 0,C 180,E1 -4876.565,E2 -4876.565} C_VEL
LIN {X 0,Y 675.766,Z 797.063,A -85,B 0,C 180,E1 -4877.337,E2 -4877.337} C_VEL
LIN {X 0,Y 675.902,Z 787.607,A -85,B 0,C 180,E1 -4878.113,E2 -4878.113} C_VEL
LIN {X 0,Y 676.042,Z 777.084,A -85,B 0,C 180,E1 -4878.813,E2 -4878.813} C_VEL
LIN {X 0,Y 676.2,Z 766.849,A -85,B 0,C 180,E1 -4879.358,E2 -4879.358} C_VEL
LIN {X 0,Y 676.348,Z 755.243,A -85,B 0,C 180,E1 -4879.847,E2 -4879.847} C_VEL
LIN {X 0,Y 676.459,Z 742.266,A -85,B 0,C 180,E1 -4880.257,E2 -4880.257} C_VEL
LIN {X 0,Y 676.636,Z 729.554,A -85,B 0,C 180,E1 -4880.528,E2 -4880.528} C_VEL
LIN {X 0,Y 676.757,Z 704.472,A -85,B 0,C 180,E1 -4880.821,E2 -4880.821} C_VEL
LIN {X 0,Y 676.789,Z 627.758,A -85,B 0,C 180,E1 -4881.634,E2 -4881.634} C_VEL
LIN {X 0,Y 675.797,Z 620.701,A -85,B 0,C 180,E1 -4881.738,E2 -4881.738} C_VEL
LIN {X 0,Y 676.025,Z 603.056,A -85,B 0,C 180,E1 -4884.484,E2 -4884.484} C_VEL
LIN {X 0,Y 676.16,Z 594.582,A -85,B 0,C 180,E1 -4885.816,E2 -4885.816} C_VEL
LIN {X 0,Y 675.565,Z 591.89,A -85,B 0,C 180,E1 -4886.259,E2 -4886.259} C_VEL
LIN {X 0,Y 670.013,Z 583.661,A -85,B 0,C 180,E1 -4887.725,E2 -4887.725} C_VEL
LIN {X 0,Y 669.401,Z 580.972,A -85,B 0,C 180,E1 -4888.174,E2 -4888.174} C_VEL
LIN {X 0,Y 669.098,Z 575.112,A -85,B 0,C 180,E1 -4889.129,E2 -4889.129} C_VEL
LIN {X 0,Y 668.918,Z 574.098,A -85,B 0,C 180,E1 -4889.31,E2 -4889.31} C_VEL
LIN {X 0,Y 668.935,Z 574.097,A -85,B 0,C 180,E1 -4891.988,E2 -4891.988} C_VEL
LIN {X 0,Y 668.916,Z 574.091,A -85,B 0,C 180,E1 -4894.433,E2 -4894.433} C_VEL
LIN {X 0,Y 668.895,Z 574.091,A -85,B 0,C 180,E1 -4896.647,E2 -4896.647} C_VEL
LIN {X 0,Y 668.911,Z 574.089,A -85,B 0,C 180,E1 -4899.205,E2 -4899.205} C_VEL
LIN {X 0,Y 668.912,Z 574.089,A -85,B 0,C 180,E1 -4901.276,E2 -4901.276} C_VEL
LIN {X 0,Y 668.925,Z 574.094,A -85,B 0,C 180,E1 -4903.737,E2 -4903.737} C_VEL
LIN {X 0,Y 668.931,Z 574.091,A -85,B 0,C 180,E1 -4906.283,E2 -4906.283} C_VEL
LIN {X 0,Y 668.913,Z 574.088,A -85,B 0,C 180,E1 -4908.932,E2 -4908.932} C_VEL
LIN {X 0,Y 668.888,Z 574.091,A -85,B 0,C 180,E1 -4911.075,E2 -4911.075} C_VEL
LIN {X 0,Y 668.899,Z 574.097,A -85,B 0,C 180,E1 -4913.737,E2 -4913.737} C_VEL
LIN {X 0,Y 668.905,Z 574.094,A -85,B 0,C 180,E1 -4916.29,E2 -4916.29} C_VEL
LIN {X 0,Y 668.913,Z 574.091,A -85,B 0,C 180,E1 -4918.428,E2 -4918.428} C_VEL
LIN {X 0,Y 668.923,Z 574.089,A -85,B 0,C 180,E1 -4920.518,E2 -4920.518} C_VEL
LIN {X 0,Y 668.895,Z 574.091,A -85,B 0,C 180,E1 -4923.238,E2 -4923.238} C_VEL
LIN {X 0,Y 668.924,Z 574.098,A -85,B 0,C 180,E1 -4925.897,E2 -4925.897} C_VEL
LIN {X 0,Y 668.94,Z 574.087,A -85,B 0,C 180,E1 -4928.501,E2 -4928.501} C_VEL
LIN {X 0,Y 668.908,Z 574.089,A -85,B 0,C 180,E1 -4931.058,E2 -4931.058} C_VEL
LIN {X 0,Y 668.932,Z 574.09,A -85,B 0,C 180,E1 -4933.577,E2 -4933.577} C_VEL
LIN {X 0,Y 668.943,Z 574.094,A -85,B 0,C 180,E1 -4936.064,E2 -4936.064} C_VEL
LIN {X 0,Y 668.932,Z 574.088,A -85,B 0,C 180,E1 -4938.524,E2 -4938.524} C_VEL
LIN {X 0,Y 668.908,Z 574.088,A -85,B 0,C 180,E1 -4940.963,E2 -4940.963} C_VEL
LIN {X 0,Y 668.984,Z 574.081,A -85,B 0,C 180,E1 -4943.386,E2 -4943.386} C_VEL
LIN {X 0,Y 669.035,Z 574.082,A -85,B 0,C 180,E1 -4945.797,E2 -4945.797} C_VEL
LIN {X 0,Y 669.087,Z 574.066,A -85,B 0,C 180,E1 -4948.8,E2 -4948.8} C_VEL
LIN {X 0,Y 669.054,Z 574.079,A -85,B 0,C 180,E1 -4951.8,E2 -4951.8} C_VEL
LIN {X 0,Y 669.015,Z 574.075,A -85,B 0,C 180,E1 -4954.805,E2 -4954.805} C_VEL
LIN {X 0,Y 668.962,Z 574.083,A -85,B 0,C 180,E1 -4957.218,E2 -4957.218} C_VEL
LIN {X 0,Y 668.946,Z 574.091,A -85,B 0,C 180,E1 -4960.182,E2 -4960.182} C_VEL
LIN {X 0,Y 668.98,Z 574.08,A -85,B 0,C 180,E1 -4963.161,E2 -4963.161} C_VEL
LIN {X 0,Y 668.966,Z 574.09,A -85,B 0,C 180,E1 -4965.797,E2 -4965.797} C_VEL
LIN {X 0,Y 668.92,Z 574.092,A -85,B 0,C 180,E1 -4968.309,E2 -4968.309} C_VEL
LIN {X 0,Y 668.939,Z 574.085,A -85,B 0,C 180,E1 -4970.855,E2 -4970.855} C_VEL
LIN {X 0,Y 668.92,Z 574.087,A -85,B 0,C 180,E1 -4972.859,E2 -4972.859} C_VEL
LIN {X 0,Y 668.889,Z 574.094,A -85,B 0,C 180,E1 -4975.426,E2 -4975.426} C_VEL
LIN {X 0,Y 668.908,Z 574.097,A -85,B 0,C 180,E1 -4978.113,E2 -4978.113} C_VEL
LIN {X 0,Y 668.959,Z 574.082,A -85,B 0,C 180,E1 -4980.868,E2 -4980.868} C_VEL
LIN {X 0,Y 668.917,Z 574.088,A -85,B 0,C 180,E1 -4983.102,E2 -4983.102} C_VEL
LIN {X 0,Y 668.931,Z 574.097,A -85,B 0,C 180,E1 -4985.901,E2 -4985.901} C_VEL
LIN {X 0,Y 668.891,Z 574.097,A -85,B 0,C 180,E1 -4988.245,E2 -4988.245} C_VEL
LIN {X 0,Y 668.932,Z 574.088,A -85,B 0,C 180,E1 -4990.482,E2 -4990.482} C_VEL
LIN {X 0,Y 668.905,Z 574.089,A -85,B 0,C 180,E1 -4992.894,E2 -4992.894} C_VEL
LIN {X 0,Y 668.934,Z 574.088,A -85,B 0,C 180,E1 -4995.448,E2 -4995.448} C_VEL
LIN {X 0,Y 668.931,Z 574.096,A -85,B 0,C 180,E1 -4998.026,E2 -4998.026} C_VEL
LIN {X 0,Y 668.919,Z 574.092,A -85,B 0,C 180,E1 -5000.302,E2 -5000.302} C_VEL
LIN {X 0,Y 668.875,Z 574.093,A -85,B 0,C 180,E1 -5002.737,E2 -5002.737} C_VEL
LIN {X 0,Y 668.924,Z 574.087,A -85,B 0,C 180,E1 -5004.837,E2 -5004.837} C_VEL
LIN {X 0,Y 668.925,Z 574.094,A -85,B 0,C 180,E1 -5007.722,E2 -5007.722} C_VEL
LIN {X 0,Y 668.922,Z 574.091,A -85,B 0,C 180,E1 -5010.356,E2 -5010.356} C_VEL
LIN {X 0,Y 668.923,Z 574.087,A -85,B 0,C 180,E1 -5012.88,E2 -5012.88} C_VEL
LIN {X 0,Y 668.903,Z 574.095,A -85,B 0,C 180,E1 -5015.647,E2 -5015.647} C_VEL
LIN {X 0,Y 668.924,Z 574.097,A -85,B 0,C 180,E1 -5017.855,E2 -5017.855} C_VEL
LIN {X 0,Y 668.917,Z 574.09,A -85,B 0,C 180,E1 -5020.462,E2 -5020.462} C_VEL
LIN {X 0,Y 668.896,Z 574.09,A -85,B 0,C 180,E1 -5022.95,E2 -5022.95} C_VEL
LIN {X 0,Y 668.895,Z 574.093,A -85,B 0,C 180,E1 -5025.445,E2 -5025.445} C_VEL
LIN {X 0,Y 668.914,Z 574.099,A -85,B 0,C 180,E1 -5027.911,E2 -5027.911} C_VEL
LIN {X 0,Y 668.992,Z 574.082,A -85,B 0,C 180,E1 -5030.356,E2 -5030.356} C_VEL
LIN {X 0,Y 668.988,Z 574.081,A -85,B 0,C 180,E1 -5033.387,E2 -5033.387} C_VEL
LIN {X 0,Y 669.025,Z 574.083,A -85,B 0,C 180,E1 -5035.797,E2 -5035.797} C_VEL
LIN {X 0,Y 669.084,Z 574.067,A -85,B 0,C 180,E1 -5038.8,E2 -5038.8} C_VEL
LIN {X 0,Y 669.041,Z 574.081,A -85,B 0,C 180,E1 -5041.8,E2 -5041.8} C_VEL
LIN {X 0,Y 669.003,Z 574.077,A -85,B 0,C 180,E1 -5044.805,E2 -5044.805} C_VEL
LIN {X 0,Y 668.956,Z 574.083,A -85,B 0,C 180,E1 -5047.218,E2 -5047.218} C_VEL
LIN {X 0,Y 668.988,Z 574.085,A -85,B 0,C 180,E1 -5050.199,E2 -5050.199} C_VEL
LIN {X 0,Y 668.923,Z 574.088,A -85,B 0,C 180,E1 -5053.319,E2 -5053.319} C_VEL
LIN {X 0,Y 668.905,Z 574.098,A -85,B 0,C 180,E1 -5055.799,E2 -5055.799} C_VEL
LIN {X 0,Y 668.897,Z 574.095,A -85,B 0,C 180,E1 -5058.31,E2 -5058.31} C_VEL
LIN {X 0,Y 668.877,Z 574.092,A -85,B 0,C 180,E1 -5060.858,E2 -5060.858} C_VEL
LIN {X 0,Y 668.904,Z 574.092,A -85,B 0,C 180,E1 -5063.448,E2 -5063.448} C_VEL
LIN {X 0,Y 668.888,Z 574.1,A -85,B 0,C 180,E1 -5066.092,E2 -5066.092} C_VEL
LIN {X 0,Y 668.911,Z 574.092,A -85,B 0,C 180,E1 -5068.406,E2 -5068.406} C_VEL
LIN {X 0,Y 668.875,Z 574.093,A -85,B 0,C 180,E1 -5070.872,E2 -5070.872} C_VEL
LIN {X 0,Y 668.897,Z 574.09,A -85,B 0,C 180,E1 -5073.099,E2 -5073.099} C_VEL
LIN {X 0,Y 668.889,Z 574.102,A -85,B 0,C 180,E1 -5075.903,E2 -5075.903} C_VEL
LIN {X 0,Y 668.882,Z 574.098,A -85,B 0,C 180,E1 -5078.243,E2 -5078.243} C_VEL
LIN {X 0,Y 668.86,Z 574.097,A -85,B 0,C 180,E1 -5080.487,E2 -5080.487} C_VEL
LIN {X 0,Y 668.854,Z 574.095,A -85,B 0,C 180,E1 -5082.898,E2 -5082.898} C_VEL
LIN {X 0,Y 668.903,Z 574.092,A -85,B 0,C 180,E1 -5085.445,E2 -5085.445} C_VEL
LIN {X 0,Y 668.862,Z 574.105,A -85,B 0,C 180,E1 -5088.032,E2 -5088.032} C_VEL
LIN {X 0,Y 668.894,Z 574.091,A -85,B 0,C 180,E1 -5090.796,E2 -5090.796} C_VEL
LIN {X 0,Y 668.876,Z 574.095,A -85,B 0,C 180,E1 -5093.352,E2 -5093.352} C_VEL
LIN {X 0,Y 668.874,Z 574.102,A -85,B 0,C 180,E1 -5095.821,E2 -5095.821} C_VEL
LIN {X 0,Y 668.891,Z 574.101,A -85,B 0,C 180,E1 -5098.017,E2 -5098.017} C_VEL
LIN {X 0,Y 668.911,Z 574.09,A -85,B 0,C 180,E1 -5100.518,E2 -5100.518} C_VEL
LIN {X 0,Y 668.854,Z 574.096,A -85,B 0,C 180,E1 -5103.237,E2 -5103.237} C_VEL
LIN {X 0,Y 668.868,Z 574.102,A -85,B 0,C 180,E1 -5105.653,E2 -5105.653} C_VEL
LIN {X 0,Y 668.903,Z 574.164,A -85,B 0,C 180,E1 -5108.036,E2 -5108.036} C_VEL
LIN {X 0,Y 669.988,Z 581.015,A -85,B 0,C 180,E1 -5109.024,E2 -5109.024} C_VEL
LIN {X 0,Y 669.673,Z 599.554,A -85,B 0,C 180,E1 -5111.555,E2 -5111.555} C_VEL
LIN {X 0,Y 669.228,Z 620.372,A -85,B 0,C 180,E1 -5114.347,E2 -5114.347} C_VEL
LIN {X 0,Y 669.016,Z 637.957,A -85,B 0,C 180,E1 -5116.683,E2 -5116.683} C_VEL
LIN {X 0,Y 668.844,Z 649.332,A -85,B 0,C 180,E1 -5118.188,E2 -5118.188} C_VEL
LIN {X 0,Y 669.985,Z 658.983,A -85,B 0,C 180,E1 -5118.313,E2 -5118.313} C_VEL
LIN {X 0,Y 669.658,Z 754.913,A -85,B 0,C 180,E1 -5119.354,E2 -5119.354} C_VEL
LIN {X 0,Y 669.529,Z 765.163,A -85,B 0,C 180,E1 -5119.53,E2 -5119.53} C_VEL
LIN {X 0,Y 669.507,Z 775.6,A -85,B 0,C 180,E1 -5119.793,E2 -5119.793} C_VEL
LIN {X 0,Y 669.404,Z 785.799,A -85,B 0,C 180,E1 -5120.134,E2 -5120.134} C_VEL
LIN {X 0,Y 669.254,Z 796.38,A -85,B 0,C 180,E1 -5120.588,E2 -5120.588} C_VEL
LIN {X 0,Y 669.079,Z 806.296,A -85,B 0,C 180,E1 -5121.117,E2 -5121.117} C_VEL
LIN {X 0,Y 668.908,Z 814.565,A -85,B 0,C 180,E1 -5121.646,E2 -5121.646} C_VEL
LIN {X 0,Y 668.749,Z 823.384,A -85,B 0,C 180,E1 -5122.326,E2 -5122.326} C_VEL
LIN {X 0,Y 668.601,Z 831.489,A -85,B 0,C 180,E1 -5123.08,E2 -5123.08} C_VEL
LIN {X 0,Y 668.512,Z 838.238,A -85,B 0,C 180,E1 -5123.835,E2 -5123.835} C_VEL
LIN {X 0,Y 668.4,Z 843.881,A -85,B 0,C 180,E1 -5124.588,E2 -5124.588} C_VEL
LIN {X 0,Y 668.367,Z 849.356,A -85,B 0,C 180,E1 -5125.492,E2 -5125.492} C_VEL
LIN {X 0,Y 668.279,Z 853.656,A -85,B 0,C 180,E1 -5126.395,E2 -5126.395} C_VEL
LIN {X 0,Y 668.321,Z 855.961,A -85,B 0,C 180,E1 -5126.996,E2 -5126.996} C_VEL
LIN {X 0,Y 668.24,Z 859.18,A -85,B 0,C 180,E1 -5128.198,E2 -5128.198} C_VEL
LIN {X 0,Y 668.233,Z 860.142,A -85,B 0,C 180,E1 -5128.799,E2 -5128.799} C_VEL
LIN {X 0,Y 668.22,Z 860.999,A -85,B 0,C 180,E1 -5130,E2 -5130} C_VEL
LIN {X 0,Y 668.233,Z 860.144,A -85,B 0,C 180,E1 -5131.201,E2 -5131.201} C_VEL
LIN {X 0,Y 668.241,Z 859.183,A -85,B 0,C 180,E1 -5131.802,E2 -5131.802} C_VEL
LIN {X 0,Y 668.321,Z 855.963,A -85,B 0,C 180,E1 -5133.004,E2 -5133.004} C_VEL
LIN {X 0,Y 668.3,Z 852.388,A -85,B 0,C 180,E1 -5133.907,E2 -5133.907} C_VEL
LIN {X 0,Y 668.411,Z 846.436,A -85,B 0,C 180,E1 -5135.009,E2 -5135.009} C_VEL
LIN {X 0,Y 668.437,Z 841.751,A -85,B 0,C 180,E1 -5135.713,E2 -5135.713} C_VEL
LIN {X 0,Y 668.542,Z 835.734,A -85,B 0,C 180,E1 -5136.467,E2 -5136.467} C_VEL
LIN {X 0,Y 668.674,Z 828.476,A -85,B 0,C 180,E1 -5137.221,E2 -5137.221} C_VEL
LIN {X 0,Y 668.809,Z 819.643,A -85,B 0,C 180,E1 -5137.977,E2 -5137.977} C_VEL
LIN {X 0,Y 668.969,Z 811.177,A -85,B 0,C 180,E1 -5138.581,E2 -5138.581} C_VEL
LIN {X 0,Y 669.146,Z 800.823,A -85,B 0,C 180,E1 -5139.186,E2 -5139.186} C_VEL
LIN {X 0,Y 669.327,Z 791.329,A -85,B 0,C 180,E1 -5139.639,E2 -5139.639} C_VEL
LIN {X 0,Y 669.438,Z 780.31,A -85,B 0,C 180,E1 -5140.056,E2 -5140.056} C_VEL
LIN {X 0,Y 669.505,Z 769.456,A -85,B 0,C 180,E1 -5140.368,E2 -5140.368} C_VEL
LIN {X 0,Y 669.686,Z 759.12,A -85,B 0,C 180,E1 -5140.58,E2 -5140.58} C_VEL
LIN {X 0,Y 669.712,Z 740.695,A -85,B 0,C 180,E1 -5140.813,E2 -5140.813} C_VEL
LIN {X 0,Y 669.86,Z 657.459,A -85,B 0,C 180,E1 -5141.7,E2 -5141.7} C_VEL
LIN {X 0,Y 668.838,Z 649.147,A -85,B 0,C 180,E1 -5141.822,E2 -5141.822} C_VEL
LIN {X 0,Y 669.128,Z 629.654,A -85,B 0,C 180,E1 -5144.396,E2 -5144.396} C_VEL
LIN {X 0,Y 669.475,Z 607.476,A -85,B 0,C 180,E1 -5147.349,E2 -5147.349} C_VEL
LIN {X 0,Y 669.811,Z 588.399,A -85,B 0,C 180,E1 -5149.926,E2 -5149.926} C_VEL
LIN {X 0,Y 669.862,Z 579.624,A -85,B 0,C 180,E1 -5151.131,E2 -5151.131} C_VEL
LIN {X 0,Y 668.892,Z 574.102,A -85,B 0,C 180,E1 -5151.945,E2 -5151.945} C_VEL
LIN {X 0,Y 668.871,Z 574.097,A -85,B 0,C 180,E1 -5154.764,E2 -5154.764} C_VEL
LIN {X 0,Y 668.852,Z 574.105,A -85,B 0,C 180,E1 -5157.438,E2 -5157.438} C_VEL
LIN {X 0,Y 668.862,Z 574.101,A -85,B 0,C 180,E1 -5160.177,E2 -5160.177} C_VEL
LIN {X 0,Y 668.913,Z 574.092,A -85,B 0,C 180,E1 -5162.992,E2 -5162.992} C_VEL
LIN {X 0,Y 668.908,Z 574.095,A -85,B 0,C 180,E1 -5165.237,E2 -5165.237} C_VEL
LIN {X 0,Y 668.878,Z 574.101,A -85,B 0,C 180,E1 -5167.4,E2 -5167.4} C_VEL
LIN {X 0,Y 668.887,Z 574.098,A -85,B 0,C 180,E1 -5169.701,E2 -5169.701} C_VEL
LIN {X 0,Y 668.903,Z 574.091,A -85,B 0,C 180,E1 -5172.081,E2 -5172.081} C_VEL
LIN {X 0,Y 668.901,Z 574.092,A -85,B 0,C 180,E1 -5174.597,E2 -5174.597} C_VEL
LIN {X 0,Y 668.914,Z 574.099,A -85,B 0,C 180,E1 -5177.138,E2 -5177.138} C_VEL
LIN {X 0,Y 668.915,Z 574.09,A -85,B 0,C 180,E1 -5179.855,E2 -5179.855} C_VEL
LIN {X 0,Y 668.888,Z 574.098,A -85,B 0,C 180,E1 -5182.736,E2 -5182.736} C_VEL
LIN {X 0,Y 668.943,Z 574.094,A -85,B 0,C 180,E1 -5184.837,E2 -5184.837} C_VEL
LIN {X 0,Y 668.93,Z 574.087,A -85,B 0,C 180,E1 -5187.722,E2 -5187.722} C_VEL
LIN {X 0,Y 668.927,Z 574.091,A -85,B 0,C 180,E1 -5190.355,E2 -5190.355} C_VEL
LIN {X 0,Y 668.928,Z 574.097,A -85,B 0,C 180,E1 -5192.88,E2 -5192.88} C_VEL
LIN {X 0,Y 668.907,Z 574.091,A -85,B 0,C 180,E1 -5195.647,E2 -5195.647} C_VEL
LIN {X 0,Y 668.928,Z 574.09,A -85,B 0,C 180,E1 -5197.854,E2 -5197.854} C_VEL
LIN {X 0,Y 668.921,Z 574.101,A -85,B 0,C 180,E1 -5200.461,E2 -5200.461} C_VEL
LIN {X 0,Y 668.901,Z 574.095,A -85,B 0,C 180,E1 -5202.95,E2 -5202.95} C_VEL
LIN {X 0,Y 668.898,Z 574.093,A -85,B 0,C 180,E1 -5205.444,E2 -5205.444} C_VEL
LIN {X 0,Y 668.961,Z 574.086,A -85,B 0,C 180,E1 -5207.298,E2 -5207.298} C_VEL
LIN {X 0,Y 668.994,Z 574.09,A -85,B 0,C 180,E1 -5210.356,E2 -5210.356} C_VEL
LIN {X 0,Y 668.982,Z 574.096,A -85,B 0,C 180,E1 -5210.736,E2 -5210.736} C_VEL
LIN {X 0,Y 669.509,Z 581.036,A -85,B 0,C 180,E1 -5211.88,E2 -5211.88} C_VEL
LIN {X 0,Y 669.221,Z 597.944,A -85,B 0,C 180,E1 -5214.595,E2 -5214.595} C_VEL
LIN {X 0,Y 668.937,Z 611.217,A -85,B 0,C 180,E1 -5216.698,E2 -5216.698} C_VEL
LIN {X 0,Y 668.721,Z 621.018,A -85,B 0,C 180,E1 -5218.237,E2 -5218.237} C_VEL
LIN {X 0,Y 670.066,Z 630.76,A -85,B 0,C 180,E1 -5218.371,E2 -5218.371} C_VEL
LIN {X 0,Y 669.523,Z 726.846,A -85,B 0,C 180,E1 -5219.419,E2 -5219.419} C_VEL
LIN {X 0,Y 669.436,Z 739.434,A -85,B 0,C 180,E1 -5219.663,E2 -5219.663} C_VEL
LIN {X 0,Y 669.335,Z 752.357,A -85,B 0,C 180,E1 -5220.037,E2 -5220.037} C_VEL
LIN {X 0,Y 669.297,Z 764.506,A -85,B 0,C 180,E1 -5220.524,E2 -5220.524} C_VEL
LIN {X 0,Y 669.087,Z 776.03,A -85,B 0,C 180,E1 -5221.125,E2 -5221.125} C_VEL
LIN {X 0,Y 668.907,Z 786.37,A -85,B 0,C 180,E1 -5221.8,E2 -5221.8} C_VEL
LIN {X 0,Y 668.684,Z 794.062,A -85,B 0,C 180,E1 -5222.401,E2 -5222.401} C_VEL
LIN {X 0,Y 668.568,Z 802.021,A -85,B 0,C 180,E1 -5223.153,E2 -5223.153} C_VEL
LIN {X 0,Y 668.425,Z 808.71,A -85,B 0,C 180,E1 -5223.905,E2 -5223.905} C_VEL
LIN {X 0,Y 668.399,Z 815.204,A -85,B 0,C 180,E1 -5224.809,E2 -5224.809} C_VEL
LIN {X 0,Y 668.34,Z 820.465,A -85,B 0,C 180,E1 -5225.714,E2 -5225.714} C_VEL
LIN {X 0,Y 668.269,Z 824.508,A -85,B 0,C 180,E1 -5226.62,E2 -5226.62} C_VEL
LIN {X 0,Y 668.266,Z 826.648,A -85,B 0,C 180,E1 -5227.225,E2 -5227.225} C_VEL
LIN {X 0,Y 668.199,Z 828.341,A -85,B 0,C 180,E1 -5227.832,E2 -5227.832} C_VEL
LIN {X 0,Y 668.216,Z 829.61,A -85,B 0,C 180,E1 -5228.439,E2 -5228.439} C_VEL
LIN {X 0,Y 668.221,Z 830.478,A -85,B 0,C 180,E1 -5229.046,E2 -5229.046} C_VEL
LIN {X 0,Y 668.259,Z 831,A -85,B 0,C 180,E1 -5229.844,E2 -5229.844} C_VEL
LIN {X 0,Y 668.214,Z 830.652,A -85,B 0,C 180,E1 -5230.876,E2 -5230.876} C_VEL
LIN {X 0,Y 668.188,Z 829.891,A -85,B 0,C 180,E1 -5231.488,E2 -5231.488} C_VEL
LIN {X 0,Y 668.232,Z 828.719,A -85,B 0,C 180,E1 -5232.101,E2 -5232.101} C_VEL
LIN {X 0,Y 668.265,Z 826.549,A -85,B 0,C 180,E1 -5232.894,E2 -5232.894} C_VEL
LIN {X 0,Y 668.285,Z 822.504,A -85,B 0,C 180,E1 -5233.949,E2 -5233.949} C_VEL
LIN {X 0,Y 668.385,Z 817.721,A -85,B 0,C 180,E1 -5234.877,E2 -5234.877} C_VEL
LIN {X 0,Y 668.469,Z 811.561,A -85,B 0,C 180,E1 -5235.809,E2 -5235.809} C_VEL
LIN {X 0,Y 668.574,Z 803.833,A -85,B 0,C 180,E1 -5236.744,E2 -5236.744} C_VEL
LIN {X 0,Y 668.734,Z 794.999,A -85,B 0,C 180,E1 -5237.607,E2 -5237.607} C_VEL
LIN {X 0,Y 668.892,Z 785.046,A -85,B 0,C 180,E1 -5238.388,E2 -5238.388} C_VEL
LIN {X 0,Y 669.088,Z 773.782,A -85,B 0,C 180,E1 -5239.095,E2 -5239.095} C_VEL
LIN {X 0,Y 669.294,Z 763.074,A -85,B 0,C 180,E1 -5239.628,E2 -5239.628} C_VEL
LIN {X 0,Y 669.416,Z 751.578,A -85,B 0,C 180,E1 -5240.08,E2 -5240.08} C_VEL
LIN {X 0,Y 669.54,Z 739.135,A -85,B 0,C 180,E1 -5240.435,E2 -5240.435} C_VEL
LIN {X 0,Y 669.67,Z 726.89,A -85,B 0,C 180,E1 -5240.671,E2 -5240.671} C_VEL
LIN {X 0,Y 669.883,Z 628.789,A -85,B 0,C 180,E1 -5241.744,E2 -5241.744} C_VEL
LIN {X 0,Y 668.751,Z 620.811,A -85,B 0,C 180,E1 -5241.868,E2 -5241.868} C_VEL
LIN {X 0,Y 669.008,Z 603.876,A -85,B 0,C 180,E1 -5244.527,E2 -5244.527} C_VEL
LIN {X 0,Y 669.282,Z 587.193,A -85,B 0,C 180,E1 -5247.18,E2 -5247.18} C_VEL
LIN {X 0,Y 669.401,Z 580.972,A -85,B 0,C 180,E1 -5248.174,E2 -5248.174} C_VEL
LIN {X 0,Y 668.698,Z 579.236,A -85,B 0,C 180,E1 -5248.476,E2 -5248.476} C_VEL
LIN {X 0,Y 665.674,Z 576.813,A -85,B 0,C 180,E1 -5248.96,E2 -5248.96} C_VEL
LIN {X 0,Y 662.626,Z 575.289,A -85,B 0,C 180,E1 -5249.47,E2 -5249.47} C_VEL
LIN {X 0,Y 661.891,Z 574.975,A -85,B 0,C 180,E1 -5249.81,E2 -5249.81} C_VEL
LIN {X 0,Y 661.895,Z 574.97,A -85,B 0,C 180,E1 -5252.157,E2 -5252.157} C_VEL
LIN {X 0,Y 661.865,Z 574.966,A -85,B 0,C 180,E1 -5254.853,E2 -5254.853} C_VEL
LIN {X 0,Y 661.836,Z 574.973,A -85,B 0,C 180,E1 -5257.462,E2 -5257.462} C_VEL
LIN {X 0,Y 661.888,Z 574.967,A -85,B 0,C 180,E1 -5260.364,E2 -5260.364} C_VEL
LIN {X 0,Y 661.878,Z 574.966,A -85,B 0,C 180,E1 -5262.632,E2 -5262.632} C_VEL
LIN {X 0,Y 661.873,Z 574.965,A -85,B 0,C 180,E1 -5265.157,E2 -5265.157} C_VEL
LIN {X 0,Y 661.895,Z 574.971,A -85,B 0,C 180,E1 -5267.796,E2 -5267.796} C_VEL
LIN {X 0,Y 661.871,Z 574.967,A -85,B 0,C 180,E1 -5270.582,E2 -5270.582} C_VEL
LIN {X 0,Y 661.859,Z 574.971,A -85,B 0,C 180,E1 -5273.543,E2 -5273.543} C_VEL
LIN {X 0,Y 661.872,Z 574.976,A -85,B 0,C 180,E1 -5275.883,E2 -5275.883} C_VEL
LIN {X 0,Y 661.892,Z 574.973,A -85,B 0,C 180,E1 -5278.054,E2 -5278.054} C_VEL
LIN {X 0,Y 661.887,Z 574.97,A -85,B 0,C 180,E1 -5280.199,E2 -5280.199} C_VEL
LIN {X 0,Y 661.873,Z 574.965,A -85,B 0,C 180,E1 -5282.931,E2 -5282.931} C_VEL
LIN {X 0,Y 661.875,Z 574.97,A -85,B 0,C 180,E1 -5285.624,E2 -5285.624} C_VEL
LIN {X 0,Y 661.888,Z 574.969,A -85,B 0,C 180,E1 -5288.26,E2 -5288.26} C_VEL
LIN {X 0,Y 661.867,Z 574.966,A -85,B 0,C 180,E1 -5290.848,E2 -5290.848} C_VEL
LIN {X 0,Y 661.892,Z 574.965,A -85,B 0,C 180,E1 -5293.398,E2 -5293.398} C_VEL
LIN {X 0,Y 661.878,Z 574.966,A -85,B 0,C 180,E1 -5295.286,E2 -5295.286} C_VEL
LIN {X 0,Y 661.949,Z 574.956,A -85,B 0,C 180,E1 -5297.161,E2 -5297.161} C_VEL
LIN {X 0,Y 661.931,Z 574.964,A -85,B 0,C 180,E1 -5300.252,E2 -5300.252} C_VEL
LIN {X 0,Y 661.924,Z 574.959,A -85,B 0,C 180,E1 -5302.705,E2 -5302.705} C_VEL
LIN {X 0,Y 661.985,Z 574.951,A -85,B 0,C 180,E1 -5305.144,E2 -5305.144} C_VEL
LIN {X 0,Y 662.044,Z 574.944,A -85,B 0,C 180,E1 -5308.787,E2 -5308.787} C_VEL
LIN {X 0,Y 662.023,Z 574.955,A -85,B 0,C 180,E1 -5311.819,E2 -5311.819} C_VEL
LIN {X 0,Y 661.985,Z 574.951,A -85,B 0,C 180,E1 -5314.856,E2 -5314.856} C_VEL
LIN {X 0,Y 661.923,Z 574.96,A -85,B 0,C 180,E1 -5317.295,E2 -5317.295} C_VEL
LIN {X 0,Y 661.909,Z 574.967,A -85,B 0,C 180,E1 -5320.22,E2 -5320.22} C_VEL
LIN {X 0,Y 661.949,Z 574.956,A -85,B 0,C 180,E1 -5323.222,E2 -5323.222} C_VEL
LIN {X 0,Y 661.906,Z 574.973,A -85,B 0,C 180,E1 -5325.97,E2 -5325.97} C_VEL
LIN {X 0,Y 661.868,Z 574.968,A -85,B 0,C 180,E1 -5328.511,E2 -5328.511} C_VEL
LIN {X 0,Y 661.906,Z 574.961,A -85,B 0,C 180,E1 -5331.088,E2 -5331.088} C_VEL
LIN {X 0,Y 661.869,Z 574.973,A -85,B 0,C 180,E1 -5333.712,E2 -5333.712} C_VEL
LIN {X 0,Y 661.832,Z 574.974,A -85,B 0,C 180,E1 -5336.391,E2 -5336.391} C_VEL
LIN {X 0,Y 661.884,Z 574.964,A -85,B 0,C 180,E1 -5339.13,E2 -5339.13} C_VEL
LIN {X 0,Y 661.892,Z 574.964,A -85,B 0,C 180,E1 -5341.234,E2 -5341.234} C_VEL
LIN {X 0,Y 661.872,Z 574.968,A -85,B 0,C 180,E1 -5343.388,E2 -5343.388} C_VEL
LIN {X 0,Y 661.891,Z 574.968,A -85,B 0,C 180,E1 -5345.594,E2 -5345.594} C_VEL
LIN {X 0,Y 661.851,Z 574.971,A -85,B 0,C 180,E1 -5348.451,E2 -5348.451} C_VEL
LIN {X 0,Y 661.88,Z 574.966,A -85,B 0,C 180,E1 -5351.292,E2 -5351.292} C_VEL
LIN {X 0,Y 661.869,Z 574.977,A -85,B 0,C 180,E1 -5353.976,E2 -5353.976} C_VEL
LIN {X 0,Y 661.881,Z 574.966,A -85,B 0,C 180,E1 -5356.539,E2 -5356.539} C_VEL
LIN {X 0,Y 661.881,Z 574.964,A -85,B 0,C 180,E1 -5358.996,E2 -5358.996} C_VEL
LIN {X 0,Y 661.853,Z 574.972,A -85,B 0,C 180,E1 -5361.55,E2 -5361.55} C_VEL
LIN {X 0,Y 661.887,Z 574.965,A -85,B 0,C 180,E1 -5364.573,E2 -5364.573} C_VEL
LIN {X 0,Y 661.865,Z 574.968,A -85,B 0,C 180,E1 -5367.335,E2 -5367.335} C_VEL
LIN {X 0,Y 661.888,Z 574.967,A -85,B 0,C 180,E1 -5369.472,E2 -5369.472} C_VEL
LIN {X 0,Y 661.877,Z 574.969,A -85,B 0,C 180,E1 -5371.562,E2 -5371.562} C_VEL
LIN {X 0,Y 661.855,Z 574.973,A -85,B 0,C 180,E1 -5374.285,E2 -5374.285} C_VEL
LIN {X 0,Y 661.899,Z 574.962,A -85,B 0,C 180,E1 -5377.023,E2 -5377.023} C_VEL
LIN {X 0,Y 661.864,Z 574.971,A -85,B 0,C 180,E1 -5379.56,E2 -5379.56} C_VEL
LIN {X 0,Y 661.903,Z 574.967,A -85,B 0,C 180,E1 -5382.252,E2 -5382.252} C_VEL
LIN {X 0,Y 661.906,Z 574.962,A -85,B 0,C 180,E1 -5384.66,E2 -5384.66} C_VEL
LIN {X 0,Y 661.928,Z 574.959,A -85,B 0,C 180,E1 -5387.161,E2 -5387.161} C_VEL
LIN {X 0,Y 661.949,Z 574.961,A -85,B 0,C 180,E1 -5390.253,E2 -5390.253} C_VEL
LIN {X 0,Y 661.949,Z 574.957,A -85,B 0,C 180,E1 -5393.316,E2 -5393.316} C_VEL
LIN {X 0,Y 661.984,Z 574.959,A -85,B 0,C 180,E1 -5395.753,E2 -5395.753} C_VEL
LIN {X 0,Y 662.043,Z 574.944,A -85,B 0,C 180,E1 -5398.788,E2 -5398.788} C_VEL
LIN {X 0,Y 662.014,Z 574.948,A -85,B 0,C 180,E1 -5401.213,E2 -5401.213} C_VEL
LIN {X 0,Y 661.972,Z 574.953,A -85,B 0,C 180,E1 -5404.856,E2 -5404.856} C_VEL
LIN {X 0,Y 661.919,Z 574.961,A -85,B 0,C 180,E1 -5407.296,E2 -5407.296} C_VEL
LIN {X 0,Y 661.945,Z 574.962,A -85,B 0,C 180,E1 -5410.235,E2 -5410.235} C_VEL
LIN {X 0,Y 661.903,Z 574.962,A -85,B 0,C 180,E1 -5413.202,E2 -5413.202} C_VEL
LIN {X 0,Y 661.865,Z 574.978,A -85,B 0,C 180,E1 -5415.971,E2 -5415.971} C_VEL
LIN {X 0,Y 661.847,Z 574.97,A -85,B 0,C 180,E1 -5418.512,E2 -5418.512} C_VEL
LIN {X 0,Y 661.837,Z 574.97,A -85,B 0,C 180,E1 -5421.09,E2 -5421.09} C_VEL
LIN {X 0,Y 661.844,Z 574.976,A -85,B 0,C 180,E1 -5423.713,E2 -5423.713} C_VEL
LIN {X 0,Y 661.848,Z 574.979,A -85,B 0,C 180,E1 -5425.899,E2 -5425.899} C_VEL
LIN {X 0,Y 661.89,Z 574.965,A -85,B 0,C 180,E1 -5428.557,E2 -5428.557} C_VEL
LIN {X 0,Y 661.816,Z 574.973,A -85,B 0,C 180,E1 -5431.238,E2 -5431.238} C_VEL
LIN {X 0,Y 661.859,Z 574.969,A -85,B 0,C 180,E1 -5433.389,E2 -5433.389} C_VEL
LIN {X 0,Y 661.843,Z 574.973,A -85,B 0,C 180,E1 -5436.346,E2 -5436.346} C_VEL
LIN {X 0,Y 661.839,Z 574.97,A -85,B 0,C 180,E1 -5438.639,E2 -5438.639} C_VEL
LIN {X 0,Y 661.847,Z 574.97,A -85,B 0,C 180,E1 -5441.288,E2 -5441.288} C_VEL
LIN {X 0,Y 661.841,Z 574.974,A -85,B 0,C 180,E1 -5444.306,E2 -5444.306} C_VEL
LIN {X 0,Y 661.807,Z 574.973,A -85,B 0,C 180,E1 -5446.91,E2 -5446.91} C_VEL
LIN {X 0,Y 661.83,Z 574.976,A -85,B 0,C 180,E1 -5449.641,E2 -5449.641} C_VEL
LIN {X 0,Y 661.829,Z 574.979,A -85,B 0,C 180,E1 -5452.132,E2 -5452.132} C_VEL
LIN {X 0,Y 661.851,Z 574.969,A -85,B 0,C 180,E1 -5454.577,E2 -5454.577} C_VEL
LIN {X 0,Y 661.839,Z 574.971,A -85,B 0,C 180,E1 -5457.334,E2 -5457.334} C_VEL
LIN {X 0,Y 661.839,Z 574.977,A -85,B 0,C 180,E1 -5460.171,E2 -5460.171} C_VEL
LIN {X 0,Y 661.833,Z 574.97,A -85,B 0,C 180,E1 -5462.93,E2 -5462.93} C_VEL
LIN {X 0,Y 661.833,Z 574.978,A -85,B 0,C 180,E1 -5465.622,E2 -5465.622} C_VEL
LIN {X 0,Y 661.863,Z 575.098,A -85,B 0,C 180,E1 -5467.933,E2 -5467.933} C_VEL
LIN {X 0,Y 663.005,Z 582.055,A -85,B 0,C 180,E1 -5468.949,E2 -5468.949} C_VEL
LIN {X 0,Y 662.688,Z 599.448,A -85,B 0,C 180,E1 -5471.353,E2 -5471.353} C_VEL
LIN {X 0,Y 662.252,Z 619.241,A -85,B 0,C 180,E1 -5474.038,E2 -5474.038} C_VEL
LIN {X 0,Y 661.969,Z 637.84,A -85,B 0,C 180,E1 -5476.539,E2 -5476.539} C_VEL
LIN {X 0,Y 661.799,Z 649.118,A -85,B 0,C 180,E1 -5478.051,E2 -5478.051} C_VEL
LIN {X 0,Y 663.049,Z 660.166,A -85,B 0,C 180,E1 -5478.209,E2 -5478.209} C_VEL
LIN {X 0,Y 662.711,Z 754.304,A -85,B 0,C 180,E1 -5479.243,E2 -5479.243} C_VEL
LIN {X 0,Y 662.549,Z 764.998,A -85,B 0,C 180,E1 -5479.427,E2 -5479.427} C_VEL
LIN {X 0,Y 662.522,Z 775.158,A -85,B 0,C 180,E1 -5479.685,E2 -5479.685} C_VEL
LIN {X 0,Y 662.385,Z 785.418,A -85,B 0,C 180,E1 -5480.029,E2 -5480.029} C_VEL
LIN {X 0,Y 662.233,Z 796.043,A -85,B 0,C 180,E1 -5480.487,E2 -5480.487} C_VEL
LIN {X 0,Y 662.015,Z 805.991,A -85,B 0,C 180,E1 -5481.022,E2 -5481.022} C_VEL
LIN {X 0,Y 661.848,Z 815.311,A -85,B 0,C 180,E1 -5481.633,E2 -5481.633} C_VEL
LIN {X 0,Y 661.686,Z 823.131,A -85,B 0,C 180,E1 -5482.243,E2 -5482.243} C_VEL
LIN {X 0,Y 661.552,Z 831.257,A -85,B 0,C 180,E1 -5483.006,E2 -5483.006} C_VEL
LIN {X 0,Y 661.434,Z 838.024,A -85,B 0,C 180,E1 -5483.769,E2 -5483.769} C_VEL
LIN {X 0,Y 661.328,Z 844.25,A -85,B 0,C 180,E1 -5484.621,E2 -5484.621} C_VEL
LIN {X 0,Y 661.288,Z 849.169,A -85,B 0,C 180,E1 -5485.444,E2 -5485.444} C_VEL
LIN {X 0,Y 661.191,Z 853.48,A -85,B 0,C 180,E1 -5486.356,E2 -5486.356} C_VEL
LIN {X 0,Y 661.22,Z 855.788,A -85,B 0,C 180,E1 -5486.964,E2 -5486.964} C_VEL
LIN {X 0,Y 661.157,Z 859.019,A -85,B 0,C 180,E1 -5488.179,E2 -5488.179} C_VEL
LIN {X 0,Y 661.16,Z 860.549,A -85,B 0,C 180,E1 -5489.393,E2 -5489.393} C_VEL
LIN {X 0,Y 661.148,Z 860.843,A -85,B 0,C 180,E1 -5490,E2 -5490} C_VEL
LIN {X 0,Y 661.14,Z 859.982,A -85,B 0,C 180,E1 -5491.214,E2 -5491.214} C_VEL
LIN {X 0,Y 661.157,Z 859.018,A -85,B 0,C 180,E1 -5491.821,E2 -5491.821} C_VEL
LIN {X 0,Y 661.221,Z 855.782,A -85,B 0,C 180,E1 -5493.036,E2 -5493.036} C_VEL
LIN {X 0,Y 661.222,Z 852.194,A -85,B 0,C 180,E1 -5493.948,E2 -5493.948} C_VEL
LIN {X 0,Y 661.31,Z 847.491,A -85,B 0,C 180,E1 -5494.861,E2 -5494.861} C_VEL
LIN {X 0,Y 661.368,Z 841.521,A -85,B 0,C 180,E1 -5495.775,E2 -5495.775} C_VEL
LIN {X 0,Y 661.447,Z 835.481,A -85,B 0,C 180,E1 -5496.537,E2 -5496.537} C_VEL
LIN {X 0,Y 661.614,Z 828.197,A -85,B 0,C 180,E1 -5497.299,E2 -5497.299} C_VEL
LIN {X 0,Y 661.762,Z 819.334,A -85,B 0,C 180,E1 -5498.062,E2 -5498.062} C_VEL
LIN {X 0,Y 661.94,Z 810.831,A -85,B 0,C 180,E1 -5498.673,E2 -5498.673} C_VEL
LIN {X 0,Y 662.132,Z 800.433,A -85,B 0,C 180,E1 -5499.284,E2 -5499.284} C_VEL
LIN {X 0,Y 662.301,Z 790.877,A -85,B 0,C 180,E1 -5499.742,E2 -5499.742} C_VEL
LIN {X 0,Y 662.432,Z 780.988,A -85,B 0,C 180,E1 -5500.125,E2 -5500.125} C_VEL
LIN {X 0,Y 662.507,Z 769.381,A -85,B 0,C 180,E1 -5500.465,E2 -5500.465} C_VEL
LIN {X 0,Y 662.688,Z 759.202,A -85,B 0,C 180,E1 -5500.679,E2 -5500.679} C_VEL
LIN {X 0,Y 662.712,Z 739.55,A -85,B 0,C 180,E1 -5500.929,E2 -5500.929} C_VEL
LIN {X 0,Y 662.94,Z 658.167,A -85,B 0,C 180,E1 -5501.813,E2 -5501.813} C_VEL
LIN {X 0,Y 661.77,Z 648.96,A -85,B 0,C 180,E1 -5501.95,E2 -5501.95} C_VEL
LIN {X 0,Y 662.075,Z 630.628,A -85,B 0,C 180,E1 -5504.396,E2 -5504.396} C_VEL
LIN {X 0,Y 662.425,Z 609.641,A -85,B 0,C 180,E1 -5507.222,E2 -5507.222} C_VEL
LIN {X 0,Y 662.83,Z 591.011,A -85,B 0,C 180,E1 -5509.765,E2 -5509.765} C_VEL
LIN {X 0,Y 662.943,Z 581.726,A -85,B 0,C 180,E1 -5511.053,E2 -5511.053} C_VEL
LIN {X 0,Y 661.842,Z 574.98,A -85,B 0,C 180,E1 -5512.068,E2 -5512.068} C_VEL
LIN {X 0,Y 661.843,Z 574.973,A -85,B 0,C 180,E1 -5515.045,E2 -5515.045} C_VEL
LIN {X 0,Y 661.818,Z 574.986,A -85,B 0,C 180,E1 -5517.754,E2 -5517.754} C_VEL
LIN {X 0,Y 661.84,Z 574.981,A -85,B 0,C 180,E1 -5519.829,E2 -5519.829} C_VEL
LIN {X 0,Y 661.847,Z 574.971,A -85,B 0,C 180,E1 -5522.666,E2 -5522.666} C_VEL
LIN {X 0,Y 661.879,Z 574.974,A -85,B 0,C 180,E1 -5525.426,E2 -5525.426} C_VEL
LIN {X 0,Y 661.837,Z 574.974,A -85,B 0,C 180,E1 -5527.867,E2 -5527.867} C_VEL
LIN {X 0,Y 661.842,Z 574.968,A -85,B 0,C 180,E1 -5530.36,E2 -5530.36} C_VEL
LIN {X 0,Y 661.872,Z 574.966,A -85,B 0,C 180,E1 -5532.633,E2 -5532.633} C_VEL
LIN {X 0,Y 661.867,Z 574.976,A -85,B 0,C 180,E1 -5535.158,E2 -5535.158} C_VEL
LIN {X 0,Y 661.899,Z 574.966,A -85,B 0,C 180,E1 -5537.797,E2 -5537.797} C_VEL
LIN {X 0,Y 661.875,Z 574.969,A -85,B 0,C 180,E1 -5540.583,E2 -5540.583} C_VEL
LIN {X 0,Y 661.895,Z 574.965,A -85,B 0,C 180,E1 -5543.657,E2 -5543.657} C_VEL
LIN {X 0,Y 661.879,Z 574.966,A -85,B 0,C 180,E1 -5545.883,E2 -5545.883} C_VEL
LIN {X 0,Y 661.884,Z 574.974,A -85,B 0,C 180,E1 -5548.765,E2 -5548.765} C_VEL
LIN {X 0,Y 661.895,Z 574.965,A -85,B 0,C 180,E1 -5551.443,E2 -5551.443} C_VEL
LIN {X 0,Y 661.852,Z 574.972,A -85,B 0,C 180,E1 -5554.101,E2 -5554.101} C_VEL
LIN {X 0,Y 661.901,Z 574.97,A -85,B 0,C 180,E1 -5556.949,E2 -5556.949} C_VEL
LIN {X 0,Y 661.868,Z 574.969,A -85,B 0,C 180,E1 -5559.559,E2 -5559.559} C_VEL
LIN {X 0,Y 661.907,Z 574.972,A -85,B 0,C 180,E1 -5562.251,E2 -5562.251} C_VEL
LIN {X 0,Y 661.909,Z 574.97,A -85,B 0,C 180,E1 -5564.659,E2 -5564.659} C_VEL
LIN {X 0,Y 661.94,Z 574.961,A -85,B 0,C 180,E1 -5567.161,E2 -5567.161} C_VEL
LIN {X 0,Y 661.952,Z 574.968,A -85,B 0,C 180,E1 -5570.253,E2 -5570.253} C_VEL
LIN {X 0,Y 661.984,Z 575.18,A -85,B 0,C 180,E1 -5570.676,E2 -5570.676} C_VEL
LIN {X 0,Y 662.524,Z 581.873,A -85,B 0,C 180,E1 -5571.794,E2 -5571.794} C_VEL
LIN {X 0,Y 662.214,Z 598.799,A -85,B 0,C 180,E1 -5574.537,E2 -5574.537} C_VEL
LIN {X 0,Y 661.912,Z 612.086,A -85,B 0,C 180,E1 -5576.663,E2 -5576.663} C_VEL
LIN {X 0,Y 661.685,Z 621.172,A -85,B 0,C 180,E1 -5578.104,E2 -5578.104} C_VEL
LIN {X 0,Y 663.097,Z 630.269,A -85,B 0,C 180,E1 -5578.241,E2 -5578.241} C_VEL
LIN {X 0,Y 662.53,Z 727.01,A -85,B 0,C 180,E1 -5579.318,E2 -5579.318} C_VEL
LIN {X 0,Y 662.447,Z 738.795,A -85,B 0,C 180,E1 -5579.545,E2 -5579.545} C_VEL
LIN {X 0,Y 662.358,Z 749.586,A -85,B 0,C 180,E1 -5579.848,E2 -5579.848} C_VEL
LIN {X 0,Y 662.295,Z 759.856,A -85,B 0,C 180,E1 -5580.227,E2 -5580.227} C_VEL
LIN {X 0,Y 662.202,Z 769.614,A -85,B 0,C 180,E1 -5580.682,E2 -5580.682} C_VEL
LIN {X 0,Y 662.026,Z 778.998,A -85,B 0,C 180,E1 -5581.212,E2 -5581.212} C_VEL
LIN {X 0,Y 661.862,Z 787.814,A -85,B 0,C 180,E1 -5581.819,E2 -5581.819} C_VEL
LIN {X 0,Y 661.611,Z 795.313,A -85,B 0,C 180,E1 -5582.427,E2 -5582.427} C_VEL
LIN {X 0,Y 661.489,Z 803.094,A -85,B 0,C 180,E1 -5583.187,E2 -5583.187} C_VEL
LIN {X 0,Y 661.326,Z 809.633,A -85,B 0,C 180,E1 -5583.947,E2 -5583.947} C_VEL
LIN {X 0,Y 661.308,Z 815.995,A -85,B 0,C 180,E1 -5584.861,E2 -5584.861} C_VEL
LIN {X 0,Y 661.251,Z 821.515,A -85,B 0,C 180,E1 -5585.86,E2 -5585.86} C_VEL
LIN {X 0,Y 661.199,Z 826.182,A -85,B 0,C 180,E1 -5586.997,E2 -5586.997} C_VEL
LIN {X 0,Y 661.101,Z 828.76,A -85,B 0,C 180,E1 -5587.917,E2 -5587.917} C_VEL
LIN {X 0,Y 661.134,Z 830.758,A -85,B 0,C 180,E1 -5589.144,E2 -5589.144} C_VEL
LIN {X 0,Y 661.161,Z 831.161,A -85,B 0,C 180,E1 -5589.85,E2 -5589.85} C_VEL
LIN {X 0,Y 661.131,Z 830.704,A -85,B 0,C 180,E1 -5590.994,E2 -5590.994} C_VEL
LIN {X 0,Y 661.134,Z 828.604,A -85,B 0,C 180,E1 -5592.233,E2 -5592.233} C_VEL
LIN {X 0,Y 661.179,Z 826.678,A -85,B 0,C 180,E1 -5592.931,E2 -5592.931} C_VEL
LIN {X 0,Y 661.214,Z 822.118,A -85,B 0,C 180,E1 -5594.102,E2 -5594.102} C_VEL
LIN {X 0,Y 661.312,Z 817.171,A -85,B 0,C 180,E1 -5595.04,E2 -5595.04} C_VEL
LIN {X 0,Y 661.376,Z 810.842,A -85,B 0,C 180,E1 -5595.983,E2 -5595.983} C_VEL
LIN {X 0,Y 661.498,Z 804.316,A -85,B 0,C 180,E1 -5596.77,E2 -5596.77} C_VEL
LIN {X 0,Y 661.658,Z 797.311,A -85,B 0,C 180,E1 -5597.482,E2 -5597.482} C_VEL
LIN {X 0,Y 661.826,Z 788.864,A -85,B 0,C 180,E1 -5598.192,E2 -5598.192} C_VEL
LIN {X 0,Y 661.924,Z 779.816,A -85,B 0,C 180,E1 -5598.829,E2 -5598.829} C_VEL
LIN {X 0,Y 662.107,Z 770.265,A -85,B 0,C 180,E1 -5599.378,E2 -5599.378} C_VEL
LIN {X 0,Y 662.326,Z 759.963,A -85,B 0,C 180,E1 -5599.861,E2 -5599.861} C_VEL
LIN {X 0,Y 662.407,Z 749.06,A -85,B 0,C 180,E1 -5600.261,E2 -5600.261} C_VEL
LIN {X 0,Y 662.567,Z 738.28,A -85,B 0,C 180,E1 -5600.559,E2 -5600.559} C_VEL
LIN {X 0,Y 662.687,Z 726.784,A -85,B 0,C 180,E1 -5600.778,E2 -5600.778} C_VEL
LIN {X 0,Y 662.975,Z 629.688,A -85,B 0,C 180,E1 -5601.858,E2 -5601.858} C_VEL
LIN {X 0,Y 661.71,Z 620.984,A -85,B 0,C 180,E1 -5601.991,E2 -5601.991} C_VEL
LIN {X 0,Y 662.008,Z 603.718,A -85,B 0,C 180,E1 -5604.731,E2 -5604.731} C_VEL
LIN {X 0,Y 662.303,Z 587.501,A -85,B 0,C 180,E1 -5607.33,E2 -5607.33} C_VEL
LIN {X 0,Y 662.36,Z 578.193,A -85,B 0,C 180,E1 -5608.839,E2 -5608.839} C_VEL
LIN {X 0,Y 661.896,Z 574.973,A -85,B 0,C 180,E1 -5609.39,E2 -5609.39} C_VEL
LIN {X 0,Y 661.891,Z 574.975,A -85,B 0,C 180,E1 -5609.81,E2 -5609.81} C_VEL
LIN {X 0,Y 661.233,Z 575.058,A -85,B 0,C 180,E1 -5610.318,E2 -5610.318} C_VEL
LIN {X 0,Y 658.394,Z 575.411,A -85,B 0,C 180,E1 -5611.142,E2 -5611.142} C_VEL
LIN {X 0,Y 655.982,Z 575.71,A -85,B 0,C 180,E1 -5611.805,E2 -5611.805} C_VEL
LIN {X 0,Y 654.929,Z 575.835,A -85,B 0,C 180,E1 -5612.316,E2 -5612.316} C_VEL
LIN {X 0,Y 654.834,Z 575.844,A -85,B 0,C 180,E1 -5612.489,E2 -5612.489} C_VEL
LIN {X 0,Y 654.832,Z 575.843,A -85,B 0,C 180,E1 -5615.282,E2 -5615.282} C_VEL
LIN {X 0,Y 654.81,Z 575.851,A -85,B 0,C 180,E1 -5617.667,E2 -5617.667} C_VEL
LIN {X 0,Y 654.855,Z 575.841,A -85,B 0,C 180,E1 -5620.586,E2 -5620.586} C_VEL
LIN {X 0,Y 654.826,Z 575.845,A -85,B 0,C 180,E1 -5623.333,E2 -5623.333} C_VEL
LIN {X 0,Y 654.825,Z 575.855,A -85,B 0,C 180,E1 -5625.95,E2 -5625.95} C_VEL
LIN {X 0,Y 654.848,Z 575.843,A -85,B 0,C 180,E1 -5628.481,E2 -5628.481} C_VEL
LIN {X 0,Y 654.806,Z 575.845,A -85,B 0,C 180,E1 -5630.867,E2 -5630.867} C_VEL
LIN {X 0,Y 654.822,Z 575.845,A -85,B 0,C 180,E1 -5633.345,E2 -5633.345} C_VEL
LIN {X 0,Y 654.825,Z 575.846,A -85,B 0,C 180,E1 -5635.464,E2 -5635.464} C_VEL
LIN {X 0,Y 654.847,Z 575.846,A -85,B 0,C 180,E1 -5637.672,E2 -5637.672} C_VEL
LIN {X 0,Y 654.848,Z 575.842,A -85,B 0,C 180,E1 -5640.526,E2 -5640.526} C_VEL
LIN {X 0,Y 654.813,Z 575.846,A -85,B 0,C 180,E1 -5643.303,E2 -5643.303} C_VEL
LIN {X 0,Y 654.836,Z 575.852,A -85,B 0,C 180,E1 -5646.017,E2 -5646.017} C_VEL
LIN {X 0,Y 654.847,Z 575.841,A -85,B 0,C 180,E1 -5648.674,E2 -5648.674} C_VEL
LIN {X 0,Y 654.828,Z 575.844,A -85,B 0,C 180,E1 -5651.283,E2 -5651.283} C_VEL
LIN {X 0,Y 654.859,Z 575.848,A -85,B 0,C 180,E1 -5653.853,E2 -5653.853} C_VEL
LIN {X 0,Y 654.902,Z 575.834,A -85,B 0,C 180,E1 -5656.723,E2 -5656.723} C_VEL
LIN {X 0,Y 654.864,Z 575.846,A -85,B 0,C 180,E1 -5659.745,E2 -5659.745} C_VEL
LIN {X 0,Y 654.898,Z 575.835,A -85,B 0,C 180,E1 -5662.626,E2 -5662.626} C_VEL
LIN {X 0,Y 654.956,Z 575.827,A -85,B 0,C 180,E1 -5665.092,E2 -5665.092} C_VEL
LIN {X 0,Y 655.005,Z 575.821,A -85,B 0,C 180,E1 -5668.774,E2 -5668.774} C_VEL
LIN {X 0,Y 655.005,Z 575.821,A -85,B 0,C 180,E1 -5671.225,E2 -5671.225} C_VEL
LIN {X 0,Y 654.956,Z 575.827,A -85,B 0,C 180,E1 -5674.908,E2 -5674.908} C_VEL
LIN {X 0,Y 654.898,Z 575.836,A -85,B 0,C 180,E1 -5677.374,E2 -5677.374} C_VEL
LIN {X 0,Y 654.863,Z 575.844,A -85,B 0,C 180,E1 -5680.255,E2 -5680.255} C_VEL
LIN {X 0,Y 654.901,Z 575.835,A -85,B 0,C 180,E1 -5683.276,E2 -5683.276} C_VEL
LIN {X 0,Y 654.859,Z 575.847,A -85,B 0,C 180,E1 -5686.147,E2 -5686.147} C_VEL
LIN {X 0,Y 654.839,Z 575.842,A -85,B 0,C 180,E1 -5688.717,E2 -5688.717} C_VEL
LIN {X 0,Y 654.867,Z 575.841,A -85,B 0,C 180,E1 -5691.481,E2 -5691.481} C_VEL
LIN {X 0,Y 654.836,Z 575.853,A -85,B 0,C 180,E1 -5693.983,E2 -5693.983} C_VEL
LIN {X 0,Y 654.812,Z 575.845,A -85,B 0,C 180,E1 -5696.697,E2 -5696.697} C_VEL
LIN {X 0,Y 654.85,Z 575.843,A -85,B 0,C 180,E1 -5699.474,E2 -5699.474} C_VEL
LIN {X 0,Y 654.838,Z 575.847,A -85,B 0,C 180,E1 -5701.609,E2 -5701.609} C_VEL
LIN {X 0,Y 654.821,Z 575.852,A -85,B 0,C 180,E1 -5703.795,E2 -5703.795} C_VEL
LIN {X 0,Y 654.821,Z 575.854,A -85,B 0,C 180,E1 -5706.038,E2 -5706.038} C_VEL
LIN {X 0,Y 654.805,Z 575.846,A -85,B 0,C 180,E1 -5708.66,E2 -5708.66} C_VEL
LIN {X 0,Y 654.851,Z 575.84,A -85,B 0,C 180,E1 -5710.728,E2 -5710.728} C_VEL
LIN {X 0,Y 654.823,Z 575.845,A -85,B 0,C 180,E1 -5713.334,E2 -5713.334} C_VEL
LIN {X 0,Y 654.823,Z 575.855,A -85,B 0,C 180,E1 -5715.951,E2 -5715.951} C_VEL
LIN {X 0,Y 654.847,Z 575.843,A -85,B 0,C 180,E1 -5718.481,E2 -5718.481} C_VEL
LIN {X 0,Y 654.807,Z 575.845,A -85,B 0,C 180,E1 -5720.868,E2 -5720.868} C_VEL
LIN {X 0,Y 654.816,Z 575.846,A -85,B 0,C 180,E1 -5723.346,E2 -5723.346} C_VEL
LIN {X 0,Y 654.826,Z 575.846,A -85,B 0,C 180,E1 -5725.465,E2 -5725.465} C_VEL
LIN {X 0,Y 654.848,Z 575.846,A -85,B 0,C 180,E1 -5727.673,E2 -5727.673} C_VEL
LIN {X 0,Y 654.849,Z 575.842,A -85,B 0,C 180,E1 -5730.526,E2 -5730.526} C_VEL
LIN {X 0,Y 654.815,Z 575.846,A -85,B 0,C 180,E1 -5733.304,E2 -5733.304} C_VEL
LIN {X 0,Y 654.827,Z 575.853,A -85,B 0,C 180,E1 -5736.017,E2 -5736.017} C_VEL
LIN {X 0,Y 654.85,Z 575.841,A -85,B 0,C 180,E1 -5738.674,E2 -5738.674} C_VEL
LIN {X 0,Y 654.805,Z 575.847,A -85,B 0,C 180,E1 -5741.282,E2 -5741.282} C_VEL
LIN {X 0,Y 654.83,Z 575.852,A -85,B 0,C 180,E1 -5743.853,E2 -5743.853} C_VEL
LIN {X 0,Y 654.885,Z 575.836,A -85,B 0,C 180,E1 -5747.02,E2 -5747.02} C_VEL
LIN {X 0,Y 654.914,Z 575.84,A -85,B 0,C 180,E1 -5750.147,E2 -5750.147} C_VEL
LIN {X 0,Y 654.899,Z 575.835,A -85,B 0,C 180,E1 -5752.626,E2 -5752.626} C_VEL
LIN {X 0,Y 654.856,Z 575.842,A -85,B 0,C 180,E1 -5754.476,E2 -5754.476} C_VEL
LIN {X 0,Y 654.831,Z 575.847,A -85,B 0,C 180,E1 -5756.32,E2 -5756.32} C_VEL
LIN {X 0,Y 655.005,Z 575.821,A -85,B 0,C 180,E1 -5758.775,E2 -5758.775} C_VEL
LIN {X 0,Y 654.978,Z 575.825,A -85,B 0,C 180,E1 -5761.226,E2 -5761.226} C_VEL
LIN {X 0,Y 654.956,Z 575.832,A -85,B 0,C 180,E1 -5764.293,E2 -5764.293} C_VEL
LIN {X 0,Y 654.912,Z 575.833,A -85,B 0,C 180,E1 -5766.757,E2 -5766.757} C_VEL
LIN {X 0,Y 654.858,Z 575.84,A -85,B 0,C 180,E1 -5769.233,E2 -5769.233} C_VEL
LIN {X 0,Y 654.839,Z 575.841,A -85,B 0,C 180,E1 -5771.101,E2 -5771.101} C_VEL
LIN {X 0,Y 654.858,Z 575.844,A -85,B 0,C 180,E1 -5773.61,E2 -5773.61} C_VEL
LIN {X 0,Y 654.827,Z 575.85,A -85,B 0,C 180,E1 -5776.148,E2 -5776.148} C_VEL
LIN {X 0,Y 654.794,Z 575.847,A -85,B 0,C 180,E1 -5778.718,E2 -5778.718} C_VEL
LIN {X 0,Y 654.796,Z 575.85,A -85,B 0,C 180,E1 -5781.464,E2 -5781.464} C_VEL
LIN {X 0,Y 654.813,Z 575.856,A -85,B 0,C 180,E1 -5783.984,E2 -5783.984} C_VEL
LIN {X 0,Y 654.816,Z 575.845,A -85,B 0,C 180,E1 -5786.697,E2 -5786.697} C_VEL
LIN {X 0,Y 654.827,Z 575.846,A -85,B 0,C 180,E1 -5789.475,E2 -5789.475} C_VEL
LIN {X 0,Y 654.82,Z 575.848,A -85,B 0,C 180,E1 -5792.333,E2 -5792.333} C_VEL
LIN {X 0,Y 654.806,Z 575.847,A -85,B 0,C 180,E1 -5794.546,E2 -5794.546} C_VEL
LIN {X 0,Y 654.777,Z 575.849,A -85,B 0,C 180,E1 -5796.802,E2 -5796.802} C_VEL
LIN {X 0,Y 654.781,Z 575.849,A -85,B 0,C 180,E1 -5799.135,E2 -5799.135} C_VEL
LIN {X 0,Y 654.793,Z 575.852,A -85,B 0,C 180,E1 -5801.546,E2 -5801.546} C_VEL
LIN {X 0,Y 654.793,Z 575.853,A -85,B 0,C 180,E1 -5804.216,E2 -5804.216} C_VEL
LIN {X 0,Y 654.772,Z 575.85,A -85,B 0,C 180,E1 -5806.793,E2 -5806.793} C_VEL
LIN {X 0,Y 654.788,Z 575.851,A -85,B 0,C 180,E1 -5809.421,E2 -5809.421} C_VEL
LIN {X 0,Y 654.814,Z 575.851,A -85,B 0,C 180,E1 -5811.653,E2 -5811.653} C_VEL
LIN {X 0,Y 654.812,Z 575.848,A -85,B 0,C 180,E1 -5814.386,E2 -5814.386} C_VEL
LIN {X 0,Y 654.8,Z 575.846,A -85,B 0,C 180,E1 -5816.938,E2 -5816.938} C_VEL
LIN {X 0,Y 654.791,Z 575.848,A -85,B 0,C 180,E1 -5819.105,E2 -5819.105} C_VEL
LIN {X 0,Y 654.796,Z 575.848,A -85,B 0,C 180,E1 -5821.302,E2 -5821.302} C_VEL
LIN {X 0,Y 654.796,Z 575.858,A -85,B 0,C 180,E1 -5823.987,E2 -5823.987} C_VEL
LIN {X 0,Y 654.796,Z 575.858,A -85,B 0,C 180,E1 -5826.015,E2 -5826.015} C_VEL
LIN {X 0,Y 654.812,Z 575.887,A -85,B 0,C 180,E1 -5827.807,E2 -5827.807} C_VEL
LIN {X 0,Y 656.017,Z 583.135,A -85,B 0,C 180,E1 -5828.878,E2 -5828.878} C_VEL
LIN {X 0,Y 655.718,Z 599.342,A -85,B 0,C 180,E1 -5831.148,E2 -5831.148} C_VEL
LIN {X 0,Y 655.274,Z 619.136,A -85,B 0,C 180,E1 -5833.864,E2 -5833.864} C_VEL
LIN {X 0,Y 654.938,Z 636.539,A -85,B 0,C 180,E1 -5836.234,E2 -5836.234} C_VEL
LIN {X 0,Y 654.752,Z 648.977,A -85,B 0,C 180,E1 -5837.92,E2 -5837.92} C_VEL
LIN {X 0,Y 656.085,Z 661.515,A -85,B 0,C 180,E1 -5838.101,E2 -5838.101} C_VEL
LIN {X 0,Y 655.728,Z 753.731,A -85,B 0,C 180,E1 -5839.129,E2 -5839.129} C_VEL
LIN {X 0,Y 655.569,Z 764.783,A -85,B 0,C 180,E1 -5839.321,E2 -5839.321} C_VEL
LIN {X 0,Y 655.53,Z 774.974,A -85,B 0,C 180,E1 -5839.582,E2 -5839.582} C_VEL
LIN {X 0,Y 655.376,Z 785.037,A -85,B 0,C 180,E1 -5839.921,E2 -5839.921} C_VEL
LIN {X 0,Y 655.215,Z 795.706,A -85,B 0,C 180,E1 -5840.385,E2 -5840.385} C_VEL
LIN {X 0,Y 655.007,Z 805.689,A -85,B 0,C 180,E1 -5840.925,E2 -5840.925} C_VEL
LIN {X 0,Y 654.794,Z 815.035,A -85,B 0,C 180,E1 -5841.542,E2 -5841.542} C_VEL
LIN {X 0,Y 654.621,Z 822.879,A -85,B 0,C 180,E1 -5842.159,E2 -5842.159} C_VEL
LIN {X 0,Y 654.477,Z 831.024,A -85,B 0,C 180,E1 -5842.93,E2 -5842.93} C_VEL
LIN {X 0,Y 654.347,Z 837.808,A -85,B 0,C 180,E1 -5843.701,E2 -5843.701} C_VEL
LIN {X 0,Y 654.228,Z 843.482,A -85,B 0,C 180,E1 -5844.471,E2 -5844.471} C_VEL
LIN {X 0,Y 654.209,Z 848.983,A -85,B 0,C 180,E1 -5845.394,E2 -5845.394} C_VEL
LIN {X 0,Y 654.109,Z 853.305,A -85,B 0,C 180,E1 -5846.316,E2 -5846.316} C_VEL
LIN {X 0,Y 654.119,Z 855.615,A -85,B 0,C 180,E1 -5846.931,E2 -5846.931} C_VEL
LIN {X 0,Y 654.077,Z 858.858,A -85,B 0,C 180,E1 -5848.159,E2 -5848.159} C_VEL
LIN {X 0,Y 654.064,Z 860.391,A -85,B 0,C 180,E1 -5849.387,E2 -5849.387} C_VEL
LIN {X 0,Y 654.052,Z 860.684,A -85,B 0,C 180,E1 -5850,E2 -5850} C_VEL
LIN {X 0,Y 654.051,Z 859.819,A -85,B 0,C 180,E1 -5851.227,E2 -5851.227} C_VEL
LIN {X 0,Y 654.077,Z 858.852,A -85,B 0,C 180,E1 -5851.841,E2 -5851.841} C_VEL
LIN {X 0,Y 654.12,Z 855.601,A -85,B 0,C 180,E1 -5853.069,E2 -5853.069} C_VEL
LIN {X 0,Y 654.148,Z 852,A -85,B 0,C 180,E1 -5853.991,E2 -5853.991} C_VEL
LIN {X 0,Y 654.212,Z 846.228,A -85,B 0,C 180,E1 -5855.083,E2 -5855.083} C_VEL
LIN {X 0,Y 654.287,Z 841.291,A -85,B 0,C 180,E1 -5855.837,E2 -5855.837} C_VEL
LIN {X 0,Y 654.384,Z 835.229,A -85,B 0,C 180,E1 -5856.608,E2 -5856.608} C_VEL
LIN {X 0,Y 654.525,Z 827.917,A -85,B 0,C 180,E1 -5857.378,E2 -5857.378} C_VEL
LIN {X 0,Y 654.7,Z 819.023,A -85,B 0,C 180,E1 -5858.15,E2 -5858.15} C_VEL
LIN {X 0,Y 654.906,Z 810.485,A -85,B 0,C 180,E1 -5858.767,E2 -5858.767} C_VEL
LIN {X 0,Y 655.063,Z 801.542,A -85,B 0,C 180,E1 -5859.307,E2 -5859.307} C_VEL
LIN {X 0,Y 655.288,Z 790.426,A -85,B 0,C 180,E1 -5859.848,E2 -5859.848} C_VEL
LIN {X 0,Y 655.408,Z 780.795,A -85,B 0,C 180,E1 -5860.223,E2 -5860.223} C_VEL
LIN {X 0,Y 655.504,Z 769.153,A -85,B 0,C 180,E1 -5860.568,E2 -5860.568} C_VEL
LIN {X 0,Y 655.689,Z 758.279,A -85,B 0,C 180,E1 -5860.794,E2 -5860.794} C_VEL
LIN {X 0,Y 655.731,Z 738.417,A -85,B 0,C 180,E1 -5861.047,E2 -5861.047} C_VEL
LIN {X 0,Y 656.01,Z 658.794,A -85,B 0,C 180,E1 -5861.93,E2 -5861.93} C_VEL
LIN {X 0,Y 654.749,Z 648.773,A -85,B 0,C 180,E1 -5862.08,E2 -5862.08} C_VEL
LIN {X 0,Y 655.071,Z 629.272,A -85,B 0,C 180,E1 -5864.712,E2 -5864.712} C_VEL
LIN {X 0,Y 655.508,Z 607.29,A -85,B 0,C 180,E1 -5867.711,E2 -5867.711} C_VEL
LIN {X 0,Y 655.883,Z 588.573,A -85,B 0,C 180,E1 -5870.309,E2 -5870.309} C_VEL
LIN {X 0,Y 655.834,Z 581.616,A -85,B 0,C 180,E1 -5871.293,E2 -5871.293} C_VEL
LIN {X 0,Y 654.788,Z 575.86,A -85,B 0,C 180,E1 -5872.153,E2 -5872.153} C_VEL
LIN {X 0,Y 654.811,Z 575.85,A -85,B 0,C 180,E1 -5874.657,E2 -5874.657} C_VEL
LIN {X 0,Y 654.792,Z 575.856,A -85,B 0,C 180,E1 -5877.394,E2 -5877.394} C_VEL
LIN {X 0,Y 654.788,Z 575.858,A -85,B 0,C 180,E1 -5879.948,E2 -5879.948} C_VEL
LIN {X 0,Y 654.821,Z 575.848,A -85,B 0,C 180,E1 -5882.333,E2 -5882.333} C_VEL
LIN {X 0,Y 654.821,Z 575.851,A -85,B 0,C 180,E1 -5885.284,E2 -5885.284} C_VEL
LIN {X 0,Y 654.81,Z 575.852,A -85,B 0,C 180,E1 -5887.668,E2 -5887.668} C_VEL
LIN {X 0,Y 654.798,Z 575.849,A -85,B 0,C 180,E1 -5889.928,E2 -5889.928} C_VEL
LIN {X 0,Y 654.824,Z 575.844,A -85,B 0,C 180,E1 -5892.433,E2 -5892.433} C_VEL
LIN {X 0,Y 654.817,Z 575.853,A -85,B 0,C 180,E1 -5895.091,E2 -5895.091} C_VEL
LIN {X 0,Y 654.847,Z 575.846,A -85,B 0,C 180,E1 -5897.634,E2 -5897.634} C_VEL
LIN {X 0,Y 654.831,Z 575.844,A -85,B 0,C 180,E1 -5900.074,E2 -5900.074} C_VEL
LIN {X 0,Y 654.812,Z 575.848,A -85,B 0,C 180,E1 -5902.431,E2 -5902.431} C_VEL
LIN {X 0,Y 654.847,Z 575.848,A -85,B 0,C 180,E1 -5904.718,E2 -5904.718} C_VEL
LIN {X 0,Y 654.853,Z 575.841,A -85,B 0,C 180,E1 -5907.672,E2 -5907.672} C_VEL
LIN {X 0,Y 654.854,Z 575.846,A -85,B 0,C 180,E1 -5910.526,E2 -5910.526} C_VEL
LIN {X 0,Y 654.819,Z 575.848,A -85,B 0,C 180,E1 -5913.303,E2 -5913.303} C_VEL
LIN {X 0,Y 654.832,Z 575.846,A -85,B 0,C 180,E1 -5916.017,E2 -5916.017} C_VEL
LIN {X 0,Y 654.854,Z 575.852,A -85,B 0,C 180,E1 -5918.674,E2 -5918.674} C_VEL
LIN {X 0,Y 654.831,Z 575.847,A -85,B 0,C 180,E1 -5921.283,E2 -5921.283} C_VEL
LIN {X 0,Y 654.834,Z 575.848,A -85,B 0,C 180,E1 -5923.852,E2 -5923.852} C_VEL
LIN {X 0,Y 654.897,Z 575.84,A -85,B 0,C 180,E1 -5927.02,E2 -5927.02} C_VEL
LIN {X 0,Y 654.916,Z 575.844,A -85,B 0,C 180,E1 -5930.147,E2 -5930.147} C_VEL
LIN {X 0,Y 654.94,Z 575.948,A -85,B 0,C 180,E1 -5930.555,E2 -5930.555} C_VEL
LIN {X 0,Y 655.541,Z 582.745,A -85,B 0,C 180,E1 -5931.706,E2 -5931.706} C_VEL
LIN {X 0,Y 655.209,Z 599.668,A -85,B 0,C 180,E1 -5934.479,E2 -5934.479} C_VEL
LIN {X 0,Y 654.89,Z 612.956,A -85,B 0,C 180,E1 -5936.627,E2 -5936.627} C_VEL
LIN {X 0,Y 654.689,Z 621.322,A -85,B 0,C 180,E1 -5937.969,E2 -5937.969} C_VEL
LIN {X 0,Y 656.155,Z 631.403,A -85,B 0,C 180,E1 -5938.126,E2 -5938.126} C_VEL
LIN {X 0,Y 655.545,Z 727.169,A -85,B 0,C 180,E1 -5939.215,E2 -5939.215} C_VEL
LIN {X 0,Y 655.466,Z 737.313,A -85,B 0,C 180,E1 -5939.407,E2 -5939.407} C_VEL
LIN {X 0,Y 655.376,Z 747.959,A -85,B 0,C 180,E1 -5939.694,E2 -5939.694} C_VEL
LIN {X 0,Y 655.307,Z 756.776,A -85,B 0,C 180,E1 -5940,E2 -5940} C_VEL
LIN {X 0,Y 655.275,Z 767.171,A -85,B 0,C 180,E1 -5940.459,E2 -5940.459} C_VEL
LIN {X 0,Y 655.043,Z 777.018,A -85,B 0,C 180,E1 -5940.995,E2 -5940.995} C_VEL
LIN {X 0,Y 654.818,Z 786.223,A -85,B 0,C 180,E1 -5941.609,E2 -5941.609} C_VEL
LIN {X 0,Y 654.57,Z 794.844,A -85,B 0,C 180,E1 -5942.3,E2 -5942.3} C_VEL
LIN {X 0,Y 654.448,Z 802.742,A -85,B 0,C 180,E1 -5943.067,E2 -5943.067} C_VEL
LIN {X 0,Y 654.27,Z 809.363,A -85,B 0,C 180,E1 -5943.836,E2 -5943.836} C_VEL
LIN {X 0,Y 654.275,Z 814.853,A -85,B 0,C 180,E1 -5944.605,E2 -5944.605} C_VEL
LIN {X 0,Y 654.15,Z 820.238,A -85,B 0,C 180,E1 -5945.53,E2 -5945.53} C_VEL
LIN {X 0,Y 654.135,Z 824.43,A -85,B 0,C 180,E1 -5946.455,E2 -5946.455} C_VEL
LIN {X 0,Y 654.063,Z 827.6,A -85,B 0,C 180,E1 -5947.383,E2 -5947.383} C_VEL
LIN {X 0,Y 654.005,Z 829.178,A -85,B 0,C 180,E1 -5948.003,E2 -5948.003} C_VEL
LIN {X 0,Y 654.053,Z 831.03,A -85,B 0,C 180,E1 -5949.244,E2 -5949.244} C_VEL
LIN {X 0,Y 654.083,Z 831.326,A -85,B 0,C 180,E1 -5949.866,E2 -5949.866} C_VEL
LIN {X 0,Y 654.022,Z 830.757,A -85,B 0,C 180,E1 -5951.115,E2 -5951.115} C_VEL
LIN {X 0,Y 654.04,Z 828.479,A -85,B 0,C 180,E1 -5952.368,E2 -5952.368} C_VEL
LIN {X 0,Y 654.097,Z 825.631,A -85,B 0,C 180,E1 -5953.311,E2 -5953.311} C_VEL
LIN {X 0,Y 654.136,Z 821.716,A -85,B 0,C 180,E1 -5954.257,E2 -5954.257} C_VEL
LIN {X 0,Y 654.25,Z 816.565,A -85,B 0,C 180,E1 -5955.206,E2 -5955.206} C_VEL
LIN {X 0,Y 654.306,Z 811.263,A -85,B 0,C 180,E1 -5956.001,E2 -5956.001} C_VEL
LIN {X 0,Y 654.42,Z 804.798,A -85,B 0,C 180,E1 -5956.797,E2 -5956.797} C_VEL
LIN {X 0,Y 654.552,Z 798.714,A -85,B 0,C 180,E1 -5957.435,E2 -5957.435} C_VEL
LIN {X 0,Y 654.758,Z 789.485,A -85,B 0,C 180,E1 -5958.234,E2 -5958.234} C_VEL
LIN {X 0,Y 654.903,Z 780.526,A -85,B 0,C 180,E1 -5958.877,E2 -5958.877} C_VEL
LIN {X 0,Y 655.069,Z 771.291,A -85,B 0,C 180,E1 -5959.422,E2 -5959.422} C_VEL
LIN {X 0,Y 655.304,Z 760.898,A -85,B 0,C 180,E1 -5959.922,E2 -5959.922} C_VEL
LIN {X 0,Y 655.428,Z 750.346,A -85,B 0,C 180,E1 -5960.323,E2 -5960.323} C_VEL
LIN {X 0,Y 655.544,Z 739.954,A -85,B 0,C 180,E1 -5960.626,E2 -5960.626} C_VEL
LIN {X 0,Y 655.683,Z 729.34,A -85,B 0,C 180,E1 -5960.846,E2 -5960.846} C_VEL
LIN {X 0,Y 655.85,Z 706.409,A -85,B 0,C 180,E1 -5961.127,E2 -5961.127} C_VEL
LIN {X 0,Y 656.063,Z 630.472,A -85,B 0,C 180,E1 -5961.976,E2 -5961.976} C_VEL
LIN {X 0,Y 654.689,Z 621.161,A -85,B 0,C 180,E1 -5962.115,E2 -5962.115} C_VEL
LIN {X 0,Y 654.993,Z 604.274,A -85,B 0,C 180,E1 -5964.818,E2 -5964.818} C_VEL
LIN {X 0,Y 655.32,Z 587.833,A -85,B 0,C 180,E1 -5967.482,E2 -5967.482} C_VEL
LIN {X 0,Y 655.394,Z 579.831,A -85,B 0,C 180,E1 -5968.793,E2 -5968.793} C_VEL
LIN {X 0,Y 654.872,Z 575.848,A -85,B 0,C 180,E1 -5969.472,E2 -5969.472} C_VEL
LIN {X 0,Y 654.85,Z 575.845,A -85,B 0,C 180,E1 -5972.331,E2 -5972.331} C_VEL
LIN {X 0,Y 654.834,Z 575.844,A -85,B 0,C 180,E1 -5972.489,E2 -5972.489} C_VEL
LIN {X 0,Y 654.141,Z 575.93,A -85,B 0,C 180,E1 -5973.002,E2 -5973.002} C_VEL
LIN {X 0,Y 651.277,Z 576.294,A -85,B 0,C 180,E1 -5973.835,E2 -5973.835} C_VEL
LIN {X 0,Y 648.879,Z 576.588,A -85,B 0,C 180,E1 -5974.505,E2 -5974.505} C_VEL
LIN {X 0,Y 647.859,Z 576.711,A -85,B 0,C 180,E1 -5975.022,E2 -5975.022} C_VEL
LIN {X 0,Y 647.781,Z 576.721,A -85,B 0,C 180,E1 -5975.197,E2 -5975.197} C_VEL
LIN {X 0,Y 647.76,Z 576.733,A -85,B 0,C 180,E1 -5977.873,E2 -5977.873} C_VEL
LIN {X 0,Y 647.814,Z 576.717,A -85,B 0,C 180,E1 -5980.811,E2 -5980.811} C_VEL
LIN {X 0,Y 647.781,Z 576.725,A -85,B 0,C 180,E1 -5983.575,E2 -5983.575} C_VEL
LIN {X 0,Y 647.78,Z 576.724,A -85,B 0,C 180,E1 -5986.424,E2 -5986.424} C_VEL
LIN {X 0,Y 647.814,Z 576.717,A -85,B 0,C 180,E1 -5989.188,E2 -5989.188} C_VEL
LIN {X 0,Y 647.76,Z 576.731,A -85,B 0,C 180,E1 -5992.126,E2 -5992.126} C_VEL
LIN {X 0,Y 647.822,Z 576.721,A -85,B 0,C 180,E1 -5994.277,E2 -5994.277} C_VEL
LIN {X 0,Y 647.787,Z 576.722,A -85,B 0,C 180,E1 -5996.533,E2 -5996.533} C_VEL
LIN {X 0,Y 647.798,Z 576.719,A -85,B 0,C 180,E1 -5998.734,E2 -5998.734} C_VEL
LIN {X 0,Y 647.819,Z 576.716,A -85,B 0,C 180,E1 -6001.139,E2 -6001.139} C_VEL
LIN {X 0,Y 647.763,Z 576.732,A -85,B 0,C 180,E1 -6003.83,E2 -6003.83} C_VEL
LIN {X 0,Y 647.811,Z 576.72,A -85,B 0,C 180,E1 -6006.418,E2 -6006.418} C_VEL
LIN {X 0,Y 647.786,Z 576.72,A -85,B 0,C 180,E1 -6009.094,E2 -6009.094} C_VEL
LIN {X 0,Y 647.797,Z 576.726,A -85,B 0,C 180,E1 -6011.725,E2 -6011.725} C_VEL
LIN {X 0,Y 647.849,Z 576.717,A -85,B 0,C 180,E1 -6014.318,E2 -6014.318} C_VEL
LIN {X 0,Y 647.862,Z 576.71,A -85,B 0,C 180,E1 -6016.877,E2 -6016.877} C_VEL
LIN {X 0,Y 647.826,Z 576.722,A -85,B 0,C 180,E1 -6019.706,E2 -6019.706} C_VEL
LIN {X 0,Y 647.853,Z 576.713,A -85,B 0,C 180,E1 -6022.545,E2 -6022.545} C_VEL
LIN {X 0,Y 647.929,Z 576.702,A -85,B 0,C 180,E1 -6025.038,E2 -6025.038} C_VEL
LIN {X 0,Y 647.969,Z 576.697,A -85,B 0,C 180,E1 -6028.761,E2 -6028.761} C_VEL
LIN {X 0,Y 647.969,Z 576.698,A -85,B 0,C 180,E1 -6031.239,E2 -6031.239} C_VEL
LIN {X 0,Y 647.929,Z 576.702,A -85,B 0,C 180,E1 -6034.961,E2 -6034.961} C_VEL
LIN {X 0,Y 647.853,Z 576.715,A -85,B 0,C 180,E1 -6037.455,E2 -6037.455} C_VEL
LIN {X 0,Y 647.826,Z 576.72,A -85,B 0,C 180,E1 -6040.294,E2 -6040.294} C_VEL
LIN {X 0,Y 647.851,Z 576.714,A -85,B 0,C 180,E1 -6043.331,E2 -6043.331} C_VEL
LIN {X 0,Y 647.817,Z 576.721,A -85,B 0,C 180,E1 -6046.327,E2 -6046.327} C_VEL
LIN {X 0,Y 647.811,Z 576.717,A -85,B 0,C 180,E1 -6048.928,E2 -6048.928} C_VEL
LIN {X 0,Y 647.839,Z 576.718,A -85,B 0,C 180,E1 -6051.593,E2 -6051.593} C_VEL
LIN {X 0,Y 647.775,Z 576.727,A -85,B 0,C 180,E1 -6054.261,E2 -6054.261} C_VEL
LIN {X 0,Y 647.788,Z 576.72,A -85,B 0,C 180,E1 -6057.01,E2 -6057.01} C_VEL
LIN {X 0,Y 647.81,Z 576.726,A -85,B 0,C 180,E1 -6059.826,E2 -6059.826} C_VEL
LIN {X 0,Y 647.799,Z 576.721,A -85,B 0,C 180,E1 -6062.501,E2 -6062.501} C_VEL
LIN {X 0,Y 647.781,Z 576.72,A -85,B 0,C 180,E1 -6064.966,E2 -6064.966} C_VEL
LIN {X 0,Y 647.753,Z 576.725,A -85,B 0,C 180,E1 -6067.269,E2 -6067.269} C_VEL
LIN {X 0,Y 647.789,Z 576.729,A -85,B 0,C 180,E1 -6069.852,E2 -6069.852} C_VEL
LIN {X 0,Y 647.783,Z 576.729,A -85,B 0,C 180,E1 -6072.098,E2 -6072.098} C_VEL
LIN {X 0,Y 647.785,Z 576.721,A -85,B 0,C 180,E1 -6074.655,E2 -6074.655} C_VEL
LIN {X 0,Y 647.785,Z 576.722,A -85,B 0,C 180,E1 -6077.331,E2 -6077.331} C_VEL
LIN {X 0,Y 647.808,Z 576.722,A -85,B 0,C 180,E1 -6079.553,E2 -6079.553} C_VEL
LIN {X 0,Y 647.759,Z 576.731,A -85,B 0,C 180,E1 -6082.127,E2 -6082.127} C_VEL
LIN {X 0,Y 647.814,Z 576.722,A -85,B 0,C 180,E1 -6084.277,E2 -6084.277} C_VEL
LIN {X 0,Y 647.787,Z 576.722,A -85,B 0,C 180,E1 -6086.533,E2 -6086.533} C_VEL
LIN {X 0,Y 647.799,Z 576.719,A -85,B 0,C 180,E1 -6088.735,E2 -6088.735} C_VEL
LIN {X 0,Y 647.82,Z 576.716,A -85,B 0,C 180,E1 -6091.14,E2 -6091.14} C_VEL
LIN {X 0,Y 647.766,Z 576.732,A -85,B 0,C 180,E1 -6093.831,E2 -6093.831} C_VEL
LIN {X 0,Y 647.784,Z 576.723,A -85,B 0,C 180,E1 -6096.417,E2 -6096.417} C_VEL
LIN {X 0,Y 647.789,Z 576.72,A -85,B 0,C 180,E1 -6099.095,E2 -6099.095} C_VEL
LIN {X 0,Y 647.783,Z 576.728,A -85,B 0,C 180,E1 -6101.725,E2 -6101.725} C_VEL
LIN {X 0,Y 647.804,Z 576.722,A -85,B 0,C 180,E1 -6104.317,E2 -6104.317} C_VEL
LIN {X 0,Y 647.831,Z 576.714,A -85,B 0,C 180,E1 -6106.877,E2 -6106.877} C_VEL
LIN {X 0,Y 647.863,Z 576.72,A -85,B 0,C 180,E1 -6110.039,E2 -6110.039} C_VEL
LIN {X 0,Y 647.855,Z 576.713,A -85,B 0,C 180,E1 -6112.546,E2 -6112.546} C_VEL
LIN {X 0,Y 647.824,Z 576.719,A -85,B 0,C 180,E1 -6114.416,E2 -6114.416} C_VEL
LIN {X 0,Y 647.806,Z 576.723,A -85,B 0,C 180,E1 -6116.281,E2 -6116.281} C_VEL
LIN {X 0,Y 647.97,Z 576.697,A -85,B 0,C 180,E1 -6118.761,E2 -6118.761} C_VEL
LIN {X 0,Y 647.945,Z 576.701,A -85,B 0,C 180,E1 -6121.239,E2 -6121.239} C_VEL
LIN {X 0,Y 647.893,Z 576.706,A -85,B 0,C 180,E1 -6124.962,E2 -6124.962} C_VEL
LIN {X 0,Y 647.852,Z 576.715,A -85,B 0,C 180,E1 -6127.455,E2 -6127.455} C_VEL
LIN {X 0,Y 647.854,Z 576.716,A -85,B 0,C 180,E1 -6130.305,E2 -6130.305} C_VEL
LIN {X 0,Y 647.822,Z 576.717,A -85,B 0,C 180,E1 -6133.318,E2 -6133.318} C_VEL
LIN {X 0,Y 647.79,Z 576.724,A -85,B 0,C 180,E1 -6136.328,E2 -6136.328} C_VEL
LIN {X 0,Y 647.772,Z 576.722,A -85,B 0,C 180,E1 -6138.929,E2 -6138.929} C_VEL
LIN {X 0,Y 647.75,Z 576.729,A -85,B 0,C 180,E1 -6141.571,E2 -6141.571} C_VEL
LIN {X 0,Y 647.76,Z 576.729,A -85,B 0,C 180,E1 -6144.262,E2 -6144.262} C_VEL
LIN {X 0,Y 647.793,Z 576.719,A -85,B 0,C 180,E1 -6147.009,E2 -6147.009} C_VEL
LIN {X 0,Y 647.787,Z 576.72,A -85,B 0,C 180,E1 -6149.116,E2 -6149.116} C_VEL
LIN {X 0,Y 647.766,Z 576.733,A -85,B 0,C 180,E1 -6151.995,E2 -6151.995} C_VEL
LIN {X 0,Y 647.765,Z 576.723,A -85,B 0,C 180,E1 -6154.734,E2 -6154.734} C_VEL
LIN {X 0,Y 647.734,Z 576.728,A -85,B 0,C 180,E1 -6157.27,E2 -6157.27} C_VEL
LIN {X 0,Y 647.754,Z 576.734,A -85,B 0,C 180,E1 -6159.848,E2 -6159.848} C_VEL
LIN {X 0,Y 647.732,Z 576.727,A -85,B 0,C 180,E1 -6162.664,E2 -6162.664} C_VEL
LIN {X 0,Y 647.761,Z 576.725,A -85,B 0,C 180,E1 -6165.343,E2 -6165.343} C_VEL
LIN {X 0,Y 647.731,Z 576.732,A -85,B 0,C 180,E1 -6168.258,E2 -6168.258} C_VEL
LIN {X 0,Y 647.757,Z 576.727,A -85,B 0,C 180,E1 -6170.358,E2 -6170.358} C_VEL
LIN {X 0,Y 647.735,Z 576.727,A -85,B 0,C 180,E1 -6173.151,E2 -6173.151} C_VEL
LIN {X 0,Y 647.734,Z 576.735,A -85,B 0,C 180,E1 -6175.784,E2 -6175.784} C_VEL
LIN {X 0,Y 647.764,Z 576.733,A -85,B 0,C 180,E1 -6178.005,E2 -6178.005} C_VEL
LIN {X 0,Y 647.751,Z 576.724,A -85,B 0,C 180,E1 -6180.882,E2 -6180.882} C_VEL
LIN {X 0,Y 647.746,Z 576.732,A -85,B 0,C 180,E1 -6183.682,E2 -6183.682} C_VEL
LIN {X 0,Y 647.748,Z 576.735,A -85,B 0,C 180,E1 -6185.738,E2 -6185.738} C_VEL
LIN {X 0,Y 647.767,Z 576.806,A -85,B 0,C 180,E1 -6187.699,E2 -6187.699} C_VEL
LIN {X 0,Y 649.029,Z 584.214,A -85,B 0,C 180,E1 -6188.805,E2 -6188.805} C_VEL
LIN {X 0,Y 648.73,Z 600.404,A -85,B 0,C 180,E1 -6191.1,E2 -6191.1} C_VEL
LIN {X 0,Y 648.251,Z 620.062,A -85,B 0,C 180,E1 -6193.828,E2 -6193.828} C_VEL
LIN {X 0,Y 647.889,Z 637.554,A -85,B 0,C 180,E1 -6196.241,E2 -6196.241} C_VEL
LIN {X 0,Y 647.728,Z 648.836,A -85,B 0,C 180,E1 -6197.787,E2 -6197.787} C_VEL
LIN {X 0,Y 649.132,Z 661.382,A -85,B 0,C 180,E1 -6197.972,E2 -6197.972} C_VEL
LIN {X 0,Y 648.736,Z 754.407,A -85,B 0,C 180,E1 -6199.032,E2 -6199.032} C_VEL
LIN {X 0,Y 648.595,Z 764.695,A -85,B 0,C 180,E1 -6199.216,E2 -6199.216} C_VEL
LIN {X 0,Y 648.53,Z 774.53,A -85,B 0,C 180,E1 -6199.468,E2 -6199.468} C_VEL
LIN {X 0,Y 648.353,Z 785.081,A -85,B 0,C 180,E1 -6199.828,E2 -6199.828} C_VEL
LIN {X 0,Y 648.216,Z 795.37,A -85,B 0,C 180,E1 -6200.28,E2 -6200.28} C_VEL
LIN {X 0,Y 647.982,Z 805.386,A -85,B 0,C 180,E1 -6200.826,E2 -6200.826} C_VEL
LIN {X 0,Y 647.736,Z 814.759,A -85,B 0,C 180,E1 -6201.449,E2 -6201.449} C_VEL
LIN {X 0,Y 647.575,Z 822.627,A -85,B 0,C 180,E1 -6202.073,E2 -6202.073} C_VEL
LIN {X 0,Y 647.424,Z 830.793,A -85,B 0,C 180,E1 -6202.853,E2 -6202.853} C_VEL
LIN {X 0,Y 647.287,Z 837.594,A -85,B 0,C 180,E1 -6203.632,E2 -6203.632} C_VEL
LIN {X 0,Y 647.161,Z 843.283,A -85,B 0,C 180,E1 -6204.41,E2 -6204.41} C_VEL
LIN {X 0,Y 647.11,Z 848.796,A -85,B 0,C 180,E1 -6205.344,E2 -6205.344} C_VEL
LIN {X 0,Y 647.031,Z 853.129,A -85,B 0,C 180,E1 -6206.276,E2 -6206.276} C_VEL
LIN {X 0,Y 647.018,Z 855.443,A -85,B 0,C 180,E1 -6206.897,E2 -6206.897} C_VEL
LIN {X 0,Y 647.001,Z 858.697,A -85,B 0,C 180,E1 -6208.139,E2 -6208.139} C_VEL
LIN {X 0,Y 646.972,Z 860.233,A -85,B 0,C 180,E1 -6209.38,E2 -6209.38} C_VEL
LIN {X 0,Y 646.96,Z 860.525,A -85,B 0,C 180,E1 -6210,E2 -6210} C_VEL
LIN {X 0,Y 646.966,Z 859.656,A -85,B 0,C 180,E1 -6211.241,E2 -6211.241} C_VEL
LIN {X 0,Y 647.002,Z 858.685,A -85,B 0,C 180,E1 -6211.861,E2 -6211.861} C_VEL
LIN {X 0,Y 647.019,Z 855.42,A -85,B 0,C 180,E1 -6213.103,E2 -6213.103} C_VEL
LIN {X 0,Y 647.076,Z 851.806,A -85,B 0,C 180,E1 -6214.035,E2 -6214.035} C_VEL
LIN {X 0,Y 647.128,Z 847.069,A -85,B 0,C 180,E1 -6214.968,E2 -6214.968} C_VEL
LIN {X 0,Y 647.215,Z 841.061,A -85,B 0,C 180,E1 -6215.901,E2 -6215.901} C_VEL
LIN {X 0,Y 647.307,Z 834.976,A -85,B 0,C 180,E1 -6216.68,E2 -6216.68} C_VEL
LIN {X 0,Y 647.467,Z 827.638,A -85,B 0,C 180,E1 -6217.459,E2 -6217.459} C_VEL
LIN {X 0,Y 647.651,Z 818.714,A -85,B 0,C 180,E1 -6218.239,E2 -6218.239} C_VEL
LIN {X 0,Y 647.872,Z 810.139,A -85,B 0,C 180,E1 -6218.863,E2 -6218.863} C_VEL
LIN {X 0,Y 648.043,Z 801.15,A -85,B 0,C 180,E1 -6219.409,E2 -6219.409} C_VEL
LIN {X 0,Y 648.253,Z 791.85,A -85,B 0,C 180,E1 -6219.877,E2 -6219.877} C_VEL
LIN {X 0,Y 648.396,Z 780.248,A -85,B 0,C 180,E1 -6220.336,E2 -6220.336} C_VEL
LIN {X 0,Y 648.506,Z 769.091,A -85,B 0,C 180,E1 -6220.669,E2 -6220.669} C_VEL
LIN {X 0,Y 648.691,Z 758.655,A -85,B 0,C 180,E1 -6220.892,E2 -6220.892} C_VEL
LIN {X 0,Y 648.744,Z 740.732,A -85,B 0,C 180,E1 -6221.128,E2 -6221.128} C_VEL
LIN {X 0,Y 649.074,Z 659.453,A -85,B 0,C 180,E1 -6222.049,E2 -6222.049} C_VEL
LIN {X 0,Y 647.724,Z 648.586,A -85,B 0,C 180,E1 -6222.213,E2 -6222.213} C_VEL
LIN {X 0,Y 648.085,Z 627.926,A -85,B 0,C 180,E1 -6225.034,E2 -6225.034} C_VEL
LIN {X 0,Y 648.502,Z 607.519,A -85,B 0,C 180,E1 -6227.858,E2 -6227.858} C_VEL
LIN {X 0,Y 649.037,Z 587.324,A -85,B 0,C 180,E1 -6230.698,E2 -6230.698} C_VEL
LIN {X 0,Y 648.679,Z 581.566,A -85,B 0,C 180,E1 -6231.539,E2 -6231.539} C_VEL
LIN {X 0,Y 647.73,Z 576.738,A -85,B 0,C 180,E1 -6232.282,E2 -6232.282} C_VEL
LIN {X 0,Y 647.772,Z 576.726,A -85,B 0,C 180,E1 -6234.943,E2 -6234.943} C_VEL
LIN {X 0,Y 647.75,Z 576.738,A -85,B 0,C 180,E1 -6237.709,E2 -6237.709} C_VEL
LIN {X 0,Y 647.736,Z 576.734,A -85,B 0,C 180,E1 -6240.106,E2 -6240.106} C_VEL
LIN {X 0,Y 647.755,Z 576.727,A -85,B 0,C 180,E1 -6242.729,E2 -6242.729} C_VEL
LIN {X 0,Y 647.81,Z 576.726,A -85,B 0,C 180,E1 -6245.724,E2 -6245.724} C_VEL
LIN {X 0,Y 647.76,Z 576.724,A -85,B 0,C 180,E1 -6248.051,E2 -6248.051} C_VEL
LIN {X 0,Y 647.773,Z 576.723,A -85,B 0,C 180,E1 -6250.807,E2 -6250.807} C_VEL
LIN {X 0,Y 647.779,Z 576.729,A -85,B 0,C 180,E1 -6253.575,E2 -6253.575} C_VEL
LIN {X 0,Y 647.784,Z 576.723,A -85,B 0,C 180,E1 -6256.425,E2 -6256.425} C_VEL
LIN {X 0,Y 647.818,Z 576.726,A -85,B 0,C 180,E1 -6259.189,E2 -6259.189} C_VEL
LIN {X 0,Y 647.764,Z 576.724,A -85,B 0,C 180,E1 -6262.127,E2 -6262.127} C_VEL
LIN {X 0,Y 647.836,Z 576.716,A -85,B 0,C 180,E1 -6264.278,E2 -6264.278} C_VEL
LIN {X 0,Y 647.793,Z 576.725,A -85,B 0,C 180,E1 -6266.533,E2 -6266.533} C_VEL
LIN {X 0,Y 647.812,Z 576.726,A -85,B 0,C 180,E1 -6268.735,E2 -6268.735} C_VEL
LIN {X 0,Y 647.825,Z 576.722,A -85,B 0,C 180,E1 -6271.139,E2 -6271.139} C_VEL
LIN {X 0,Y 647.759,Z 576.726,A -85,B 0,C 180,E1 -6273.833,E2 -6273.833} C_VEL
LIN {X 0,Y 647.812,Z 576.726,A -85,B 0,C 180,E1 -6276.418,E2 -6276.418} C_VEL
LIN {X 0,Y 647.793,Z 576.725,A -85,B 0,C 180,E1 -6279.095,E2 -6279.095} C_VEL
LIN {X 0,Y 647.794,Z 576.725,A -85,B 0,C 180,E1 -6281.725,E2 -6281.725} C_VEL
LIN {X 0,Y 647.808,Z 576.729,A -85,B 0,C 180,E1 -6284.317,E2 -6284.317} C_VEL
LIN {X 0,Y 647.842,Z 576.72,A -85,B 0,C 180,E1 -6286.876,E2 -6286.876} C_VEL
LIN {X 0,Y 647.866,Z 576.722,A -85,B 0,C 180,E1 -6290.038,E2 -6290.038} C_VEL
LIN {X 0,Y 647.901,Z 576.74,A -85,B 0,C 180,E1 -6290.432,E2 -6290.432} C_VEL
LIN {X 0,Y 648.559,Z 583.618,A -85,B 0,C 180,E1 -6291.616,E2 -6291.616} C_VEL
LIN {X 0,Y 648.207,Z 600.536,A -85,B 0,C 180,E1 -6294.419,E2 -6294.419} C_VEL
LIN {X 0,Y 647.868,Z 613.827,A -85,B 0,C 180,E1 -6296.591,E2 -6296.591} C_VEL
LIN {X 0,Y 647.702,Z 621.591,A -85,B 0,C 180,E1 -6297.85,E2 -6297.85} C_VEL
LIN {X 0,Y 649.216,Z 632.487,A -85,B 0,C 180,E1 -6298.01,E2 -6298.01} C_VEL
LIN {X 0,Y 648.576,Z 726.113,A -85,B 0,C 180,E1 -6299.091,E2 -6299.091} C_VEL
LIN {X 0,Y 648.489,Z 735.863,A -85,B 0,C 180,E1 -6299.265,E2 -6299.265} C_VEL
LIN {X 0,Y 648.398,Z 746.347,A -85,B 0,C 180,E1 -6299.536,E2 -6299.536} C_VEL
LIN {X 0,Y 648.305,Z 757.395,A -85,B 0,C 180,E1 -6299.922,E2 -6299.922} C_VEL
LIN {X 0,Y 648.266,Z 767.712,A -85,B 0,C 180,E1 -6300.387,E2 -6300.387} C_VEL
LIN {X 0,Y 648.024,Z 776.263,A -85,B 0,C 180,E1 -6300.851,E2 -6300.851} C_VEL
LIN {X 0,Y 647.82,Z 785.634,A -85,B 0,C 180,E1 -6301.471,E2 -6301.471} C_VEL
LIN {X 0,Y 647.54,Z 794.374,A -85,B 0,C 180,E1 -6302.169,E2 -6302.169} C_VEL
LIN {X 0,Y 647.401,Z 802.391,A -85,B 0,C 180,E1 -6302.946,E2 -6302.946} C_VEL
LIN {X 0,Y 647.221,Z 809.093,A -85,B 0,C 180,E1 -6303.723,E2 -6303.723} C_VEL
LIN {X 0,Y 647.18,Z 813.702,A -85,B 0,C 180,E1 -6304.345,E2 -6304.345} C_VEL
LIN {X 0,Y 647.118,Z 819.151,A -85,B 0,C 180,E1 -6305.243,E2 -6305.243} C_VEL
LIN {X 0,Y 647.072,Z 823.796,A -85,B 0,C 180,E1 -6306.214,E2 -6306.214} C_VEL
LIN {X 0,Y 647.012,Z 826.127,A -85,B 0,C 180,E1 -6306.839,E2 -6306.839} C_VEL
LIN {X 0,Y 646.913,Z 829.574,A -85,B 0,C 180,E1 -6308.091,E2 -6308.091} C_VEL
LIN {X 0,Y 646.979,Z 831.23,A -85,B 0,C 180,E1 -6309.346,E2 -6309.346} C_VEL
LIN {X 0,Y 646.989,Z 831.523,A -85,B 0,C 180,E1 -6309.975,E2 -6309.975} C_VEL
LIN {X 0,Y 646.937,Z 830.769,A -85,B 0,C 180,E1 -6311.238,E2 -6311.238} C_VEL
LIN {X 0,Y 646.934,Z 829.773,A -85,B 0,C 180,E1 -6311.871,E2 -6311.871} C_VEL
LIN {X 0,Y 647.014,Z 826.512,A -85,B 0,C 180,E1 -6313.14,E2 -6313.14} C_VEL
LIN {X 0,Y 647.048,Z 822.809,A -85,B 0,C 180,E1 -6314.097,E2 -6314.097} C_VEL
LIN {X 0,Y 647.149,Z 817.93,A -85,B 0,C 180,E1 -6315.056,E2 -6315.056} C_VEL
LIN {X 0,Y 647.222,Z 811.683,A -85,B 0,C 180,E1 -6316.019,E2 -6316.019} C_VEL
LIN {X 0,Y 647.357,Z 805.282,A -85,B 0,C 180,E1 -6316.824,E2 -6316.824} C_VEL
LIN {X 0,Y 647.549,Z 797.526,A -85,B 0,C 180,E1 -6317.63,E2 -6317.63} C_VEL
LIN {X 0,Y 647.733,Z 789.051,A -85,B 0,C 180,E1 -6318.358,E2 -6318.358} C_VEL
LIN {X 0,Y 647.868,Z 781.233,A -85,B 0,C 180,E1 -6318.926,E2 -6318.926} C_VEL
LIN {X 0,Y 648.043,Z 771.81,A -85,B 0,C 180,E1 -6319.494,E2 -6319.494} C_VEL
LIN {X 0,Y 648.296,Z 762.651,A -85,B 0,C 180,E1 -6319.951,E2 -6319.951} C_VEL
LIN {X 0,Y 648.436,Z 751.624,A -85,B 0,C 180,E1 -6320.387,E2 -6320.387} C_VEL
LIN {X 0,Y 648.537,Z 740.772,A -85,B 0,C 180,E1 -6320.714,E2 -6320.714} C_VEL
LIN {X 0,Y 648.697,Z 729.226,A -85,B 0,C 180,E1 -6320.957,E2 -6320.957} C_VEL
LIN {X 0,Y 648.848,Z 709.991,A -85,B 0,C 180,E1 -6321.201,E2 -6321.201} C_VEL
LIN {X 0,Y 649.104,Z 631.125,A -85,B 0,C 180,E1 -6322.099,E2 -6322.099} C_VEL
LIN {X 0,Y 647.683,Z 621.338,A -85,B 0,C 180,E1 -6322.241,E2 -6322.241} C_VEL
LIN {X 0,Y 647.991,Z 603.63,A -85,B 0,C 180,E1 -6325.104,E2 -6325.104} C_VEL
LIN {X 0,Y 648.343,Z 587.898,A -85,B 0,C 180,E1 -6327.681,E2 -6327.681} C_VEL
LIN {X 0,Y 648.333,Z 580.297,A -85,B 0,C 180,E1 -6328.942,E2 -6328.942} C_VEL
LIN {X 0,Y 647.841,Z 576.724,A -85,B 0,C 180,E1 -6329.557,E2 -6329.557} C_VEL
LIN {X 0,Y 647.8,Z 576.729,A -85,B 0,C 180,E1 -6331.993,E2 -6331.993} C_VEL
LIN {X 0,Y 647.785,Z 576.72,A -85,B 0,C 180,E1 -6334.736,E2 -6334.736} C_VEL
LIN {X 0,Y 647.781,Z 576.721,A -85,B 0,C 180,E1 -6335.197,E2 -6335.197} C_VEL
LIN {X 0,Y 647.126,Z 576.811,A -85,B 0,C 180,E1 -6335.716,E2 -6335.716} C_VEL
LIN {X 0,Y 644.273,Z 577.162,A -85,B 0,C 180,E1 -6336.558,E2 -6336.558} C_VEL
LIN {X 0,Y 641.851,Z 577.465,A -85,B 0,C 180,E1 -6337.236,E2 -6337.236} C_VEL
LIN {X 0,Y 640.805,Z 577.597,A -85,B 0,C 180,E1 -6337.758,E2 -6337.758} C_VEL
LIN {X 0,Y 640.717,Z 577.608,A -85,B 0,C 180,E1 -6337.935,E2 -6337.935} C_VEL
LIN {X 0,Y 640.776,Z 577.593,A -85,B 0,C 180,E1 -6340.985,E2 -6340.985} C_VEL
LIN {X 0,Y 640.755,Z 577.6,A -85,B 0,C 180,E1 -6343.526,E2 -6343.526} C_VEL
LIN {X 0,Y 640.755,Z 577.598,A -85,B 0,C 180,E1 -6346.473,E2 -6346.473} C_VEL
LIN {X 0,Y 640.776,Z 577.593,A -85,B 0,C 180,E1 -6349.014,E2 -6349.014} C_VEL
LIN {X 0,Y 640.713,Z 577.612,A -85,B 0,C 180,E1 -6351.917,E2 -6351.917} C_VEL
LIN {X 0,Y 640.773,Z 577.595,A -85,B 0,C 180,E1 -6354.595,E2 -6354.595} C_VEL
LIN {X 0,Y 640.74,Z 577.603,A -85,B 0,C 180,E1 -6357.611,E2 -6357.611} C_VEL
LIN {X 0,Y 640.77,Z 577.596,A -85,B 0,C 180,E1 -6360.534,E2 -6360.534} C_VEL
LIN {X 0,Y 640.736,Z 577.599,A -85,B 0,C 180,E1 -6362.668,E2 -6362.668} C_VEL
LIN {X 0,Y 640.742,Z 577.6,A -85,B 0,C 180,E1 -6365.455,E2 -6365.455} C_VEL
LIN {X 0,Y 640.738,Z 577.602,A -85,B 0,C 180,E1 -6367.504,E2 -6367.504} C_VEL
LIN {X 0,Y 640.776,Z 577.6,A -85,B 0,C 180,E1 -6370.192,E2 -6370.192} C_VEL
LIN {X 0,Y 640.762,Z 577.595,A -85,B 0,C 180,E1 -6372.833,E2 -6372.833} C_VEL
LIN {X 0,Y 640.775,Z 577.593,A -85,B 0,C 180,E1 -6374.79,E2 -6374.79} C_VEL
LIN {X 0,Y 640.787,Z 577.594,A -85,B 0,C 180,E1 -6377.372,E2 -6377.372} C_VEL
LIN {X 0,Y 640.787,Z 577.603,A -85,B 0,C 180,E1 -6379.927,E2 -6379.927} C_VEL
LIN {X 0,Y 640.821,Z 577.59,A -85,B 0,C 180,E1 -6382.463,E2 -6382.463} C_VEL
LIN {X 0,Y 640.881,Z 577.58,A -85,B 0,C 180,E1 -6384.984,E2 -6384.984} C_VEL
LIN {X 0,Y 640.935,Z 577.574,A -85,B 0,C 180,E1 -6388.747,E2 -6388.747} C_VEL
LIN {X 0,Y 640.935,Z 577.574,A -85,B 0,C 180,E1 -6391.252,E2 -6391.252} C_VEL
LIN {X 0,Y 640.881,Z 577.58,A -85,B 0,C 180,E1 -6395.016,E2 -6395.016} C_VEL
LIN {X 0,Y 640.821,Z 577.592,A -85,B 0,C 180,E1 -6397.537,E2 -6397.537} C_VEL
LIN {X 0,Y 640.779,Z 577.597,A -85,B 0,C 180,E1 -6400.329,E2 -6400.329} C_VEL
LIN {X 0,Y 640.805,Z 577.592,A -85,B 0,C 180,E1 -6403.389,E2 -6403.389} C_VEL
LIN {X 0,Y 640.798,Z 577.6,A -85,B 0,C 180,E1 -6405.866,E2 -6405.866} C_VEL
LIN {X 0,Y 640.757,Z 577.598,A -85,B 0,C 180,E1 -6408.482,E2 -6408.482} C_VEL
LIN {X 0,Y 640.761,Z 577.598,A -85,B 0,C 180,E1 -6410.475,E2 -6410.475} C_VEL
LIN {X 0,Y 640.789,Z 577.592,A -85,B 0,C 180,E1 -6413.173,E2 -6413.173} C_VEL
LIN {X 0,Y 640.697,Z 577.614,A -85,B 0,C 180,E1 -6415.932,E2 -6415.932} C_VEL
LIN {X 0,Y 640.773,Z 577.594,A -85,B 0,C 180,E1 -6418.749,E2 -6418.749} C_VEL
LIN {X 0,Y 640.762,Z 577.595,A -85,B 0,C 180,E1 -6420.916,E2 -6420.916} C_VEL
LIN {X 0,Y 640.735,Z 577.599,A -85,B 0,C 180,E1 -6423.134,E2 -6423.134} C_VEL
LIN {X 0,Y 640.762,Z 577.605,A -85,B 0,C 180,E1 -6426.01,E2 -6426.01} C_VEL
LIN {X 0,Y 640.729,Z 577.601,A -85,B 0,C 180,E1 -6428.544,E2 -6428.544} C_VEL
LIN {X 0,Y 640.757,Z 577.596,A -85,B 0,C 180,E1 -6431.039,E2 -6431.039} C_VEL
LIN {X 0,Y 640.753,Z 577.6,A -85,B 0,C 180,E1 -6433.526,E2 -6433.526} C_VEL
LIN {X 0,Y 640.753,Z 577.599,A -85,B 0,C 180,E1 -6436.474,E2 -6436.474} C_VEL
LIN {X 0,Y 640.774,Z 577.593,A -85,B 0,C 180,E1 -6439.015,E2 -6439.015} C_VEL
LIN {X 0,Y 640.729,Z 577.61,A -85,B 0,C 180,E1 -6441.916,E2 -6441.916} C_VEL
LIN {X 0,Y 640.768,Z 577.596,A -85,B 0,C 180,E1 -6444.595,E2 -6444.595} C_VEL
LIN {X 0,Y 640.741,Z 577.603,A -85,B 0,C 180,E1 -6447.612,E2 -6447.612} C_VEL
LIN {X 0,Y 640.771,Z 577.596,A -85,B 0,C 180,E1 -6450.534,E2 -6450.534} C_VEL
LIN {X 0,Y 640.737,Z 577.599,A -85,B 0,C 180,E1 -6452.669,E2 -6452.669} C_VEL
LIN {X 0,Y 640.74,Z 577.601,A -85,B 0,C 180,E1 -6455.455,E2 -6455.455} C_VEL
LIN {X 0,Y 640.741,Z 577.601,A -85,B 0,C 180,E1 -6457.505,E2 -6457.505} C_VEL
LIN {X 0,Y 640.779,Z 577.6,A -85,B 0,C 180,E1 -6460.193,E2 -6460.193} C_VEL
LIN {X 0,Y 640.744,Z 577.597,A -85,B 0,C 180,E1 -6462.833,E2 -6462.833} C_VEL
LIN {X 0,Y 640.739,Z 577.598,A -85,B 0,C 180,E1 -6464.79,E2 -6464.79} C_VEL
LIN {X 0,Y 640.771,Z 577.596,A -85,B 0,C 180,E1 -6467.372,E2 -6467.372} C_VEL
LIN {X 0,Y 640.813,Z 577.6,A -85,B 0,C 180,E1 -6469.928,E2 -6469.928} C_VEL
LIN {X 0,Y 640.824,Z 577.59,A -85,B 0,C 180,E1 -6472.463,E2 -6472.463} C_VEL
LIN {X 0,Y 640.797,Z 577.595,A -85,B 0,C 180,E1 -6474.354,E2 -6474.354} C_VEL
LIN {X 0,Y 640.781,Z 577.598,A -85,B 0,C 180,E1 -6476.24,E2 -6476.24} C_VEL
LIN {X 0,Y 640.937,Z 577.573,A -85,B 0,C 180,E1 -6478.748,E2 -6478.748} C_VEL
LIN {X 0,Y 640.914,Z 577.577,A -85,B 0,C 180,E1 -6481.253,E2 -6481.253} C_VEL
LIN {X 0,Y 640.862,Z 577.586,A -85,B 0,C 180,E1 -6484.388,E2 -6484.388} C_VEL
LIN {X 0,Y 640.821,Z 577.588,A -85,B 0,C 180,E1 -6486.906,E2 -6486.906} C_VEL
LIN {X 0,Y 640.82,Z 577.591,A -85,B 0,C 180,E1 -6489.437,E2 -6489.437} C_VEL
LIN {X 0,Y 640.746,Z 577.608,A -85,B 0,C 180,E1 -6491.988,E2 -6491.988} C_VEL
LIN {X 0,Y 640.778,Z 577.604,A -85,B 0,C 180,E1 -6493.915,E2 -6493.915} C_VEL
LIN {X 0,Y 640.737,Z 577.6,A -85,B 0,C 180,E1 -6496.513,E2 -6496.513} C_VEL
LIN {X 0,Y 640.719,Z 577.603,A -85,B 0,C 180,E1 -6498.484,E2 -6498.484} C_VEL
LIN {X 0,Y 640.7,Z 577.603,A -85,B 0,C 180,E1 -6501.148,E2 -6501.148} C_VEL
LIN {X 0,Y 640.718,Z 577.61,A -85,B 0,C 180,E1 -6503.859,E2 -6503.859} C_VEL
LIN {X 0,Y 640.718,Z 577.605,A -85,B 0,C 180,E1 -6506.306,E2 -6506.306} C_VEL
LIN {X 0,Y 640.774,Z 577.594,A -85,B 0,C 180,E1 -6508.749,E2 -6508.749} C_VEL
LIN {X 0,Y 640.723,Z 577.606,A -85,B 0,C 180,E1 -6511.651,E2 -6511.651} C_VEL
LIN {X 0,Y 640.711,Z 577.612,A -85,B 0,C 180,E1 -6513.886,E2 -6513.886} C_VEL
LIN {X 0,Y 640.732,Z 577.606,A -85,B 0,C 180,E1 -6516.18,E2 -6516.18} C_VEL
LIN {X 0,Y 640.714,Z 577.603,A -85,B 0,C 180,E1 -6518.546,E2 -6518.546} C_VEL
LIN {X 0,Y 640.701,Z 577.603,A -85,B 0,C 180,E1 -6521.032,E2 -6521.032} C_VEL
LIN {X 0,Y 640.712,Z 577.61,A -85,B 0,C 180,E1 -6523.819,E2 -6523.819} C_VEL
LIN {X 0,Y 640.727,Z 577.602,A -85,B 0,C 180,E1 -6526.471,E2 -6526.471} C_VEL
LIN {X 0,Y 640.704,Z 577.602,A -85,B 0,C 180,E1 -6529.009,E2 -6529.009} C_VEL
LIN {X 0,Y 640.707,Z 577.613,A -85,B 0,C 180,E1 -6531.918,E2 -6531.918} C_VEL
LIN {X 0,Y 640.717,Z 577.602,A -85,B 0,C 180,E1 -6534.591,E2 -6534.591} C_VEL
LIN {X 0,Y 640.727,Z 577.601,A -85,B 0,C 180,E1 -6537.327,E2 -6537.327} C_VEL
LIN {X 0,Y 640.708,Z 577.61,A -85,B 0,C 180,E1 -6539.809,E2 -6539.809} C_VEL
LIN {X 0,Y 640.713,Z 577.606,A -85,B 0,C 180,E1 -6542.315,E2 -6542.315} C_VEL
LIN {X 0,Y 640.748,Z 577.6,A -85,B 0,C 180,E1 -6545.138,E2 -6545.138} C_VEL
LIN {X 0,Y 640.725,Z 577.712,A -85,B 0,C 180,E1 -6547.589,E2 -6547.589} C_VEL
LIN {X 0,Y 642.056,Z 585.26,A -85,B 0,C 180,E1 -6548.732,E2 -6548.732} C_VEL
LIN {X 0,Y 641.821,Z 599.17,A -85,B 0,C 180,E1 -6550.723,E2 -6550.723} C_VEL
LIN {X 0,Y 641.264,Z 618.882,A -85,B 0,C 180,E1 -6553.501,E2 -6553.501} C_VEL
LIN {X 0,Y 640.886,Z 636.254,A -85,B 0,C 180,E1 -6555.926,E2 -6555.926} C_VEL
LIN {X 0,Y 640.702,Z 648.696,A -85,B 0,C 180,E1 -6557.651,E2 -6557.651} C_VEL
LIN {X 0,Y 642.17,Z 661.249,A -85,B 0,C 180,E1 -6557.84,E2 -6557.84} C_VEL
LIN {X 0,Y 641.752,Z 754.818,A -85,B 0,C 180,E1 -6558.929,E2 -6558.929} C_VEL
LIN {X 0,Y 641.622,Z 764.521,A -85,B 0,C 180,E1 -6559.106,E2 -6559.106} C_VEL
LIN {X 0,Y 641.511,Z 775.218,A -85,B 0,C 180,E1 -6559.389,E2 -6559.389} C_VEL
LIN {X 0,Y 641.327,Z 785.154,A -85,B 0,C 180,E1 -6559.735,E2 -6559.735} C_VEL
LIN {X 0,Y 641.202,Z 795.033,A -85,B 0,C 180,E1 -6560.172,E2 -6560.172} C_VEL
LIN {X 0,Y 640.955,Z 805.083,A -85,B 0,C 180,E1 -6560.724,E2 -6560.724} C_VEL
LIN {X 0,Y 640.702,Z 814.484,A -85,B 0,C 180,E1 -6561.355,E2 -6561.355} C_VEL
LIN {X 0,Y 640.534,Z 822.375,A -85,B 0,C 180,E1 -6561.986,E2 -6561.986} C_VEL
LIN {X 0,Y 640.355,Z 830.56,A -85,B 0,C 180,E1 -6562.774,E2 -6562.774} C_VEL
LIN {X 0,Y 640.192,Z 837.379,A -85,B 0,C 180,E1 -6563.561,E2 -6563.561} C_VEL
LIN {X 0,Y 640.095,Z 843.083,A -85,B 0,C 180,E1 -6564.348,E2 -6564.348} C_VEL
LIN {X 0,Y 640.013,Z 848.609,A -85,B 0,C 180,E1 -6565.292,E2 -6565.292} C_VEL
LIN {X 0,Y 639.957,Z 852.954,A -85,B 0,C 180,E1 -6566.235,E2 -6566.235} C_VEL
LIN {X 0,Y 639.922,Z 855.27,A -85,B 0,C 180,E1 -6566.863,E2 -6566.863} C_VEL
LIN {X 0,Y 639.929,Z 858.536,A -85,B 0,C 180,E1 -6568.118,E2 -6568.118} C_VEL
LIN {X 0,Y 639.885,Z 860.074,A -85,B 0,C 180,E1 -6569.373,E2 -6569.373} C_VEL
LIN {X 0,Y 639.872,Z 860.367,A -85,B 0,C 180,E1 -6570,E2 -6570} C_VEL
LIN {X 0,Y 639.886,Z 859.494,A -85,B 0,C 180,E1 -6571.255,E2 -6571.255} C_VEL
LIN {X 0,Y 639.929,Z 858.519,A -85,B 0,C 180,E1 -6571.882,E2 -6571.882} C_VEL
LIN {X 0,Y 639.923,Z 855.239,A -85,B 0,C 180,E1 -6573.137,E2 -6573.137} C_VEL
LIN {X 0,Y 640.006,Z 851.613,A -85,B 0,C 180,E1 -6574.079,E2 -6574.079} C_VEL
LIN {X 0,Y 640.037,Z 846.858,A -85,B 0,C 180,E1 -6575.023,E2 -6575.023} C_VEL
LIN {X 0,Y 640.145,Z 840.831,A -85,B 0,C 180,E1 -6575.967,E2 -6575.967} C_VEL
LIN {X 0,Y 640.223,Z 834.723,A -85,B 0,C 180,E1 -6576.754,E2 -6576.754} C_VEL
LIN {X 0,Y 640.407,Z 827.359,A -85,B 0,C 180,E1 -6577.542,E2 -6577.542} C_VEL
LIN {X 0,Y 640.613,Z 818.404,A -85,B 0,C 180,E1 -6578.33,E2 -6578.33} C_VEL
LIN {X 0,Y 640.818,Z 809.791,A -85,B 0,C 180,E1 -6578.961,E2 -6578.961} C_VEL
LIN {X 0,Y 641.021,Z 800.758,A -85,B 0,C 180,E1 -6579.513,E2 -6579.513} C_VEL
LIN {X 0,Y 641.245,Z 791.399,A -85,B 0,C 180,E1 -6579.986,E2 -6579.986} C_VEL
LIN {X 0,Y 641.382,Z 780.058,A -85,B 0,C 180,E1 -6580.439,E2 -6580.439} C_VEL
LIN {X 0,Y 641.52,Z 768.842,A -85,B 0,C 180,E1 -6580.777,E2 -6580.777} C_VEL
LIN {X 0,Y 641.699,Z 757.726,A -85,B 0,C 180,E1 -6581.012,E2 -6581.012} C_VEL
